% RSLogix 500 project CANHOES E PERFURATRIZES 1.RSS, saved by version 10.00.00.00 %
PROJECT "USIMINAS"    % processor: SLC 500, 1747-L552 %

PROGRAM FILES
  LAD 2 "PRINCIPAL"  17 rungs
  LAD 5 "ANA OUT"  17 rungs  % Bloco de transferencia do 1746-NO4V para o SCANNER %
  LAD 7 "BOMBA 1"  25 rungs  % Bomba 1 %
  LAD 8 "BOMBA 2"  21 rungs  % Bomba 2 %
  LAD 9 "BOMBA REF"  17 rungs  % Bomba Refrigeracao 1 %
  LAD 11 "PRESS INJ"  7 rungs  % Pressao de injecao mais alta %
  LAD 12 "TRACO INJ"  11 rungs  % Volume Lama Injetado %
  LAD 13 "CANHAO"  24 rungs  % Controle do Giro do Canhao %
  LAD 14 "INJECAO M"  10 rungs
  LAD 15 "PERFURAT"  29 rungs
  LAD 16 "MARTELETE"  10 rungs
  LAD 17 "BOMBA AGUA"  15 rungs  % Resfriamento da Broca ou Sopro %
  LAD 18 "ALR GERAIS"  69 rungs  % ALARMES GERAIS E ANUNCIADOR %
  LAD 19 "COMUNIC"  20 rungs  % Comuinicao com supervisorio - Desabilitado(futuro) %
  LAD 20 "HISTERESE"  6 rungs
  LAD 21 "ALR ANALOG"  70 rungs  % Alarmes Analogicos %
  LAD 22 "UNID ENG"  20 rungs
  LAD 23 "RESET"  10 rungs  % Reset geral para 1 scan %

DATA FILES
  O0 OUTPUT  52 elements
  I1 INPUT  46 elements
  S2 STATUS  83 elements
  B3 BINARY  63 elements
  T4 TIMER  201 elements
  C5 COUNTER  1 elements
  R6 CONTROL  4 elements
  N7 INTEGER  3 elements
  F8 FLOAT  50 elements
  B9 COMANDO D  28 elements
  B10 ESPELHO D  16 elements  % Area Espelho entradas e saidas digitais %
  B11 STATUS  68 elements  % Status do sistema que são enviados ao SSC %
  B13 DEFEITO  112 elements
  N15 ESPELHO A  50 elements  % Area Espelho entradas e saidas analogicas %
  N16 SET POINT  90 elements
  N17 LEITURA  90 elements
  N18 COMANDO A  1 elements  % Comando Analogico %
  B20 ESPELHO O  12 elements
  B21 AUXILIARES  20 elements  % auxiliares %
  B22   1 elements
  B23   1 elements
  N24 SAIDAS ANA  20 elements
  N25 B TRANSFER  10 elements  % Utilizado pelo Bloco Transfer %
  N26 COM SUP  51 elements  % Area para comunicacao com Supervisorio %
  N27 COM SUP  51 elements  % Area para comunicacao com Supervisorio %
  N29 HISTERESE  9 elements  % Valores para calculo de histerese %
  B31 AUX STATUS  26 elements
  B33 AUX DEF  26 elements
  B39 LEIT SUP  10 elements  % Area de mensagens que sao enviadas ao Supervisorio %
  B40 LEIT SUP  10 elements  % Area de mensagens que sao enviadas ao Supervisorio %
  B41 LEIT SUP  8 elements  % Area de mensagens que sao enviadas ao Supervisorio %
  B42 LEIT SUP  1 elements  % Area de mensagens que sao enviadas ao Supervisorio %

LADDER 2 "PRINCIPAL"
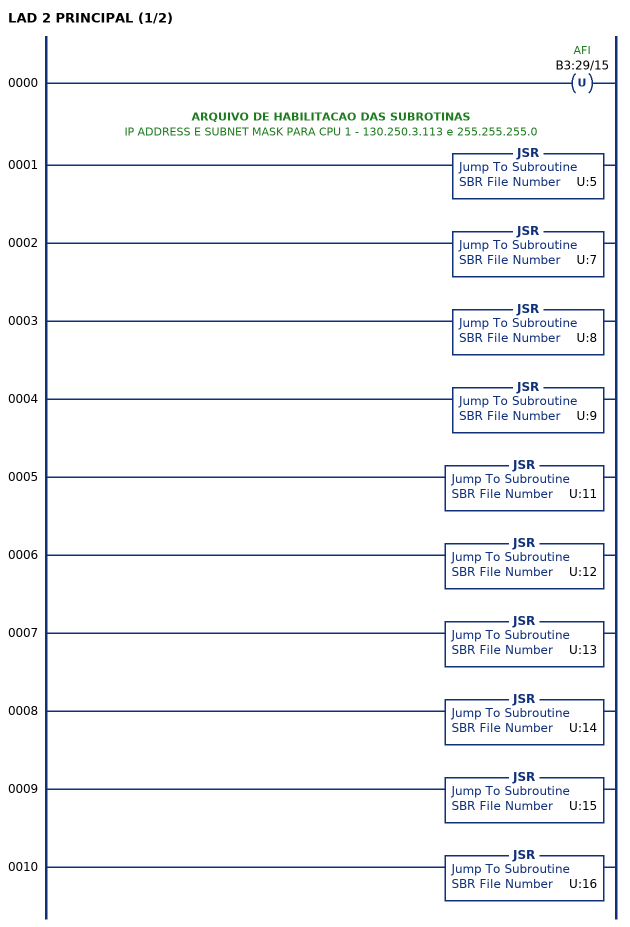
% Rung: 0 %
SOR OTU B3:29/15 EOR
%   B3:29/15  AFI %
% Rung: 1 %
% TITLE: ARQUIVO DE HABILITACAO DAS SUBROTINAS %
% IP ADDRESS E SUBNET MASK PARA CPU 1 - 130.250.3.113 e 255.255.255.0 %
SOR JSR U:5 EOR
% Rung: 2 %
SOR JSR U:7 EOR
% Rung: 3 %
SOR JSR U:8 EOR
% Rung: 4 %
SOR JSR U:9 EOR
% Rung: 5 %
SOR JSR U:11 EOR
% Rung: 6 %
SOR JSR U:12 EOR
% Rung: 7 %
SOR JSR U:13 EOR
% Rung: 8 %
SOR JSR U:14 EOR
% Rung: 9 %
SOR JSR U:15 EOR
% Rung: 10 %
SOR JSR U:16 EOR

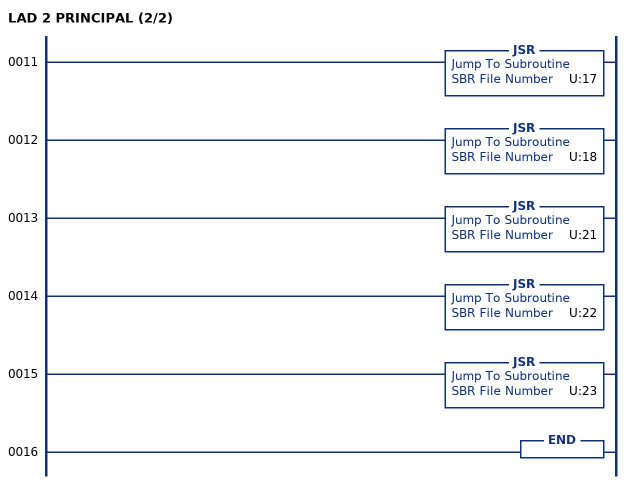
% Rung: 11 %
SOR JSR U:17 EOR
% Rung: 12 %
SOR JSR U:18 EOR
% Rung: 13 %
SOR JSR U:21 EOR
% Rung: 14 %
SOR JSR U:22 EOR
% Rung: 15 %
SOR JSR U:23 EOR
% Rung: 16 %
SOR END EOR

LADDER 5 "ANA OUT"    % Bloco de transferencia do 1746-NO4V para o SCANNER %
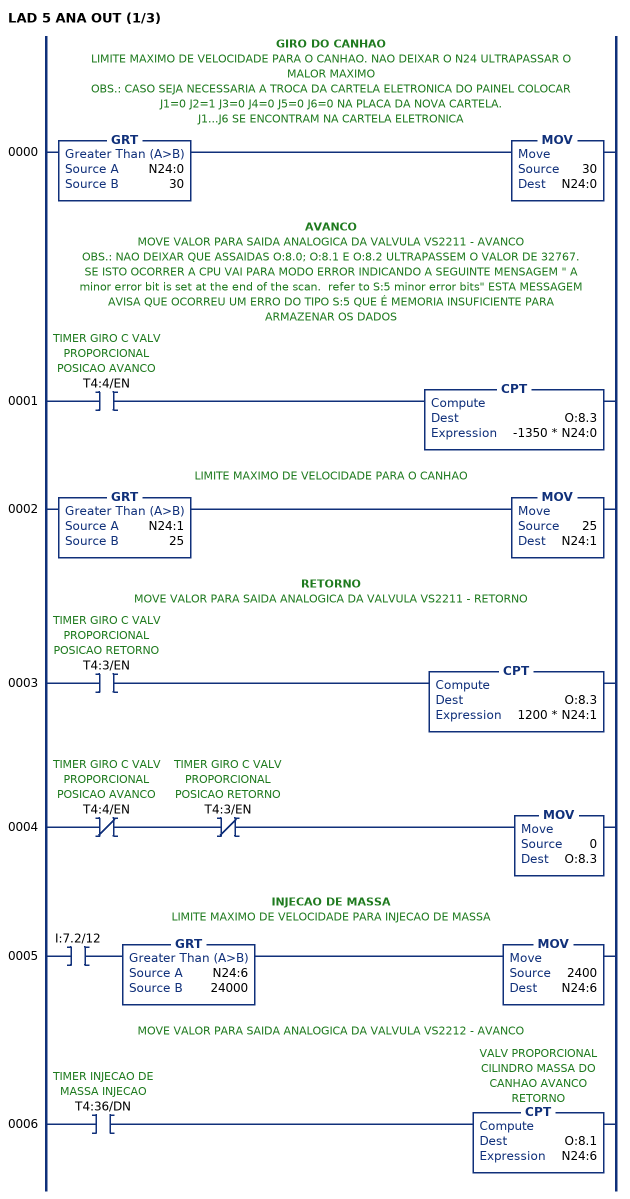
% Rung: 0 %
% TITLE: GIRO DO CANHAO %
% LIMITE MAXIMO DE VELOCIDADE PARA O CANHAO. NAO DEIXAR O N24 ULTRAPASSAR O MALOR MAXIMO
% OBS.: CASO SEJA NECESSARIA A TROCA DA CARTELA ELETRONICA DO PAINEL COLOCAR
% J1=0 J2=1 J3=0 J4=0 J5=0 J6=0 NA PLACA DA NOVA CARTELA.
% J1...J6 SE ENCONTRAM NA CARTELA ELETRONICA %
SOR GRT N24:0 30 MOV 30 N24:0 EOR
% Rung: 1 %
% TITLE: AVANCO %
% MOVE VALOR PARA SAIDA ANALOGICA DA VALVULA VS2211 - AVANCO
% OBS.: NAO DEIXAR QUE ASSAIDAS O:8.0; O:8.1 E O:8.2 ULTRAPASSEM O VALOR DE 32767. SE ISTO OCORRER A CPU VAI PARA MODO ERROR INDICANDO A SEGUINTE MENSAGEM " A minor error bit is set at the end of the scan.  refer to S:5 minor error bits" ESTA MESSAGEM AVISA QUE OCORREU UM ERRO DO TIPO S:5 QUE É MEMORIA INSUFICIENTE PARA ARMAZENAR OS DADOS %
SOR XIC T4:4/EN CPT O:8.3 " -1350 * N24:0 " EOR
%   T4:4  "TIMER GIRO C VALV PROPORCIONAL POSICAO AVANCO" %
% Rung: 2 %
% LIMITE MAXIMO DE VELOCIDADE PARA O CANHAO %
SOR GRT N24:1 25 MOV 25 N24:1 EOR
% Rung: 3 %
% TITLE: RETORNO %
% MOVE VALOR PARA SAIDA ANALOGICA DA VALVULA VS2211 - RETORNO %
SOR XIC T4:3/EN CPT O:8.3 " 1200 * N24:1 " EOR
%   T4:3  "TIMER GIRO C VALV PROPORCIONAL POSICAO RETORNO" %
% Rung: 4 %
SOR XIO T4:4/EN XIO T4:3/EN MOV 0 O:8.3 EOR
%   T4:4  "TIMER GIRO C VALV PROPORCIONAL POSICAO AVANCO" %
%   T4:3  "TIMER GIRO C VALV PROPORCIONAL POSICAO RETORNO" %
% Rung: 5 %
% TITLE: INJECAO DE MASSA %
% LIMITE MAXIMO DE VELOCIDADE PARA INJECAO DE MASSA %
SOR XIC I:7.2/12 GRT N24:6 24000 MOV 2400 N24:6 EOR
% Rung: 6 %
% MOVE VALOR PARA SAIDA ANALOGICA DA VALVULA VS2212 - AVANCO %
SOR XIC T4:36/DN CPT O:8.1 "  N24:6 " EOR
%   T4:36  "TIMER INJECAO DE MASSA INJECAO" %
%   O:8.1  "VALV PROPORCIONAL CILINDRO MASSA DO CANHAO AVANCO RETORNO" %

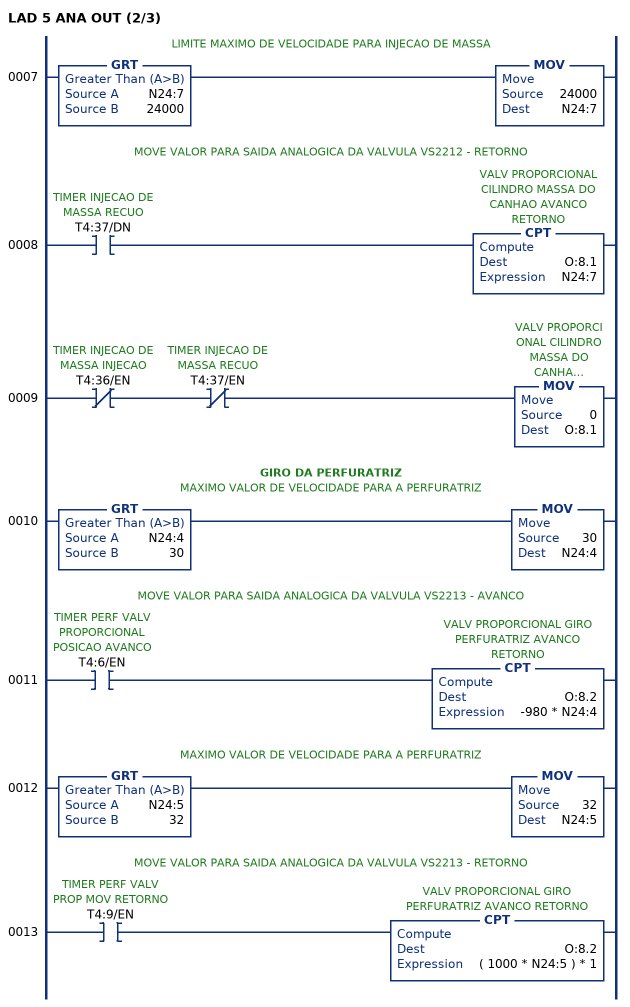
% Rung: 7 %
% LIMITE MAXIMO DE VELOCIDADE PARA INJECAO DE MASSA %
SOR GRT N24:7 24000 MOV 24000 N24:7 EOR
% Rung: 8 %
% MOVE VALOR PARA SAIDA ANALOGICA DA VALVULA VS2212 - RETORNO %
SOR XIC T4:37/DN CPT O:8.1 "  N24:7 " EOR
%   T4:37  "TIMER INJECAO DE MASSA RECUO" %
%   O:8.1  "VALV PROPORCIONAL CILINDRO MASSA DO CANHAO AVANCO RETORNO" %
% Rung: 9 %
SOR XIO T4:36/EN XIO T4:37/EN MOV 0 O:8.1 EOR
%   T4:36  "TIMER INJECAO DE MASSA INJECAO" %
%   T4:37  "TIMER INJECAO DE MASSA RECUO" %
%   O:8.1  "VALV PROPORCIONAL CILINDRO MASSA DO CANHAO AVANCO RETORNO" %
% Rung: 10 %
% TITLE: GIRO DA PERFURATRIZ %
% MAXIMO VALOR DE VELOCIDADE PARA A PERFURATRIZ %
SOR GRT N24:4 30 MOV 30 N24:4 EOR
% Rung: 11 %
% MOVE VALOR PARA SAIDA ANALOGICA DA VALVULA VS2213 - AVANCO %
SOR XIC T4:6/EN CPT O:8.2 " -980 * N24:4 " EOR
%   T4:6  "TIMER PERF VALV PROPORCIONAL POSICAO AVANCO" %
%   O:8.2  "VALV PROPORCIONAL GIRO PERFURATRIZ AVANCO RETORNO" %
% Rung: 12 %
% MAXIMO VALOR DE VELOCIDADE PARA A PERFURATRIZ %
SOR GRT N24:5 32 MOV 32 N24:5 EOR
% Rung: 13 %
% MOVE VALOR PARA SAIDA ANALOGICA DA VALVULA VS2213 - RETORNO %
SOR XIC T4:9/EN CPT O:8.2 " ( 1000 * N24:5 ) * 1 " EOR
%   T4:9  "TIMER PERF VALV PROP MOV RETORNO" %
%   O:8.2  "VALV PROPORCIONAL GIRO PERFURATRIZ AVANCO RETORNO" %

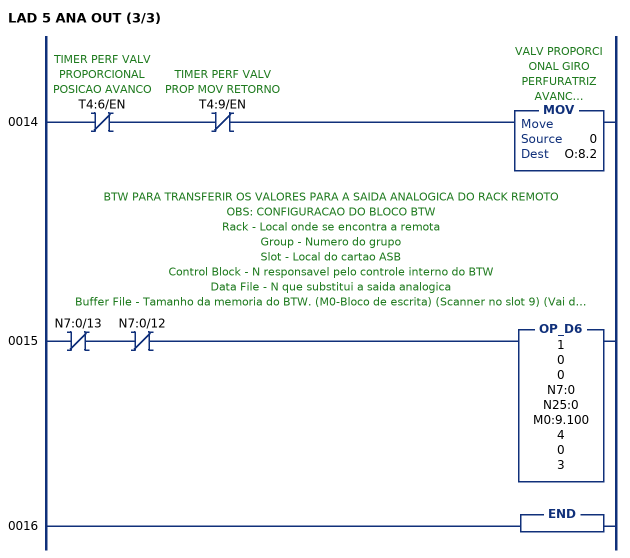
% Rung: 14 %
SOR XIO T4:6/EN XIO T4:9/EN MOV 0 O:8.2 EOR
%   T4:6  "TIMER PERF VALV PROPORCIONAL POSICAO AVANCO" %
%   T4:9  "TIMER PERF VALV PROP MOV RETORNO" %
%   O:8.2  "VALV PROPORCIONAL GIRO PERFURATRIZ AVANCO RETORNO" %
% Rung: 15 %
% BTW PARA TRANSFERIR OS VALORES PARA A SAIDA ANALOGICA DO RACK REMOTO
% OBS: CONFIGURACAO DO BLOCO BTW
% Rack - Local onde se encontra a remota
% Group - Numero do grupo
% Slot - Local do cartao ASB
% Control Block - N responsavel pelo controle interno do BTW
% Data File - N que substitui a saida analogica
% Buffer File - Tamanho da memoria do BTW. (M0-Bloco de escrita) (Scanner no slot 9) (Vai de 100 a 3200)
% Req W. C - Quantidade de palavras usadas
% Trans. W. C. - Uso interno do BTW
% Control B. L - Uso interno do BTW %
SOR XIO N7:0/13 XIO N7:0/12 OP_D6 1 0 0 N7:0 N25:0 M0:9.100 4 0 3 EOR
% Rung: 16 %
SOR END EOR

LADDER 7 "BOMBA 1"    % Bomba 1 %
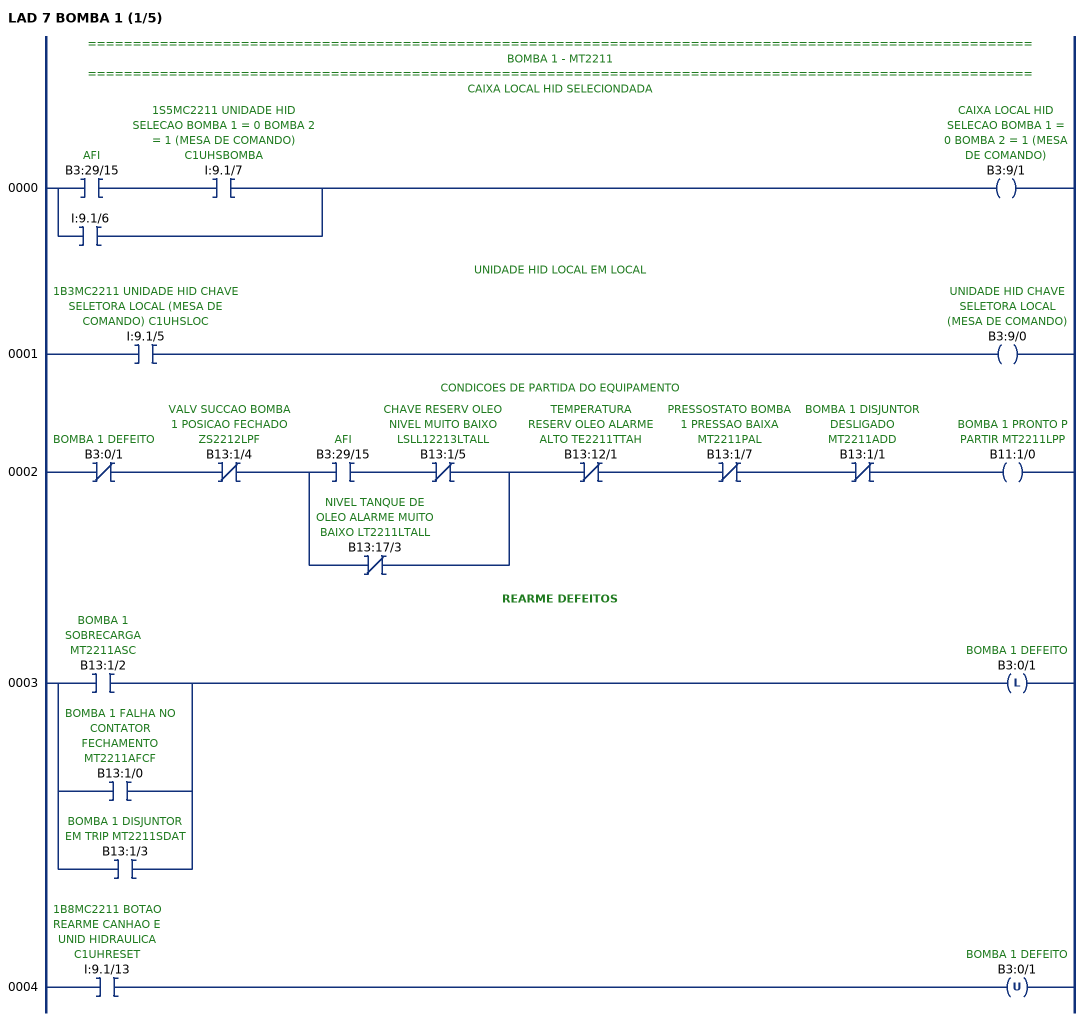
% Rung: 0 %
% =========================================================================================================
% BOMBA 1 - MT2211
% =========================================================================================================
% 
% CAIXA LOCAL HID SELECIONDADA %
SOR BST XIC B3:29/15 XIC I:9.1/7 NXB XIC I:9.1/6 BND OTE B3:9/1 EOR
%   B3:29/15  AFI %
%   I:9.1/7  C1UHSBOMBA  "1S5MC2211 UNIDADE HID SELECAO BOMBA 1 = 0 BOMBA 2 = 1 (MESA DE COMANDO)" %
%   B3:9/1  "CAIXA LOCAL HID SELECAO BOMBA 1 = 0 BOMBA 2 = 1 (MESA DE COMANDO)" %
% Rung: 1 %
% UNIDADE HID LOCAL EM LOCAL %
SOR XIC I:9.1/5 OTE B3:9/0 EOR
%   I:9.1/5  C1UHSLOC  "1B3MC2211 UNIDADE HID CHAVE SELETORA LOCAL (MESA DE COMANDO)" %
%   B3:9/0  "UNIDADE HID CHAVE SELETORA LOCAL (MESA DE COMANDO)" %
% Rung: 2 %
% CONDICOES DE PARTIDA DO EQUIPAMENTO %
SOR XIO B3:0/1 XIO B13:1/4 BST XIC B3:29/15 XIO B13:1/5 NXB XIO B13:17/3 BND XIO B13:12/1 XIO B13:1/7 XIO B13:1/1 OTE B11:1/0 EOR
%   B3:0/1  "BOMBA 1 DEFEITO" %
%   B13:1/4  ZS2212LPF  "VALV SUCCAO BOMBA 1 POSICAO FECHADO" %
%   B3:29/15  AFI %
%   B13:1/5  LSLL12213LTALL  "CHAVE RESERV OLEO NIVEL MUITO BAIXO" %
%   B13:17/3  LT2211LTALL  "NIVEL TANQUE DE OLEO ALARME MUITO BAIXO" %
%   B13:12/1  TE2211TTAH  "TEMPERATURA RESERV OLEO ALARME ALTO" %
%   B13:1/7  MT2211PAL  "PRESSOSTATO BOMBA 1 PRESSAO BAIXA" %
%   B13:1/1  MT2211ADD  "BOMBA 1 DISJUNTOR DESLIGADO" %
%   B11:1/0  MT2211LPP  "BOMBA 1 PRONTO P PARTIR" %
% Rung: 3 %
% TITLE: REARME DEFEITOS %
SOR BST XIC B13:1/2 NXB XIC B13:1/0 NXB XIC B13:1/3 BND OTL B3:0/1 EOR
%   B13:1/2  MT2211ASC  "BOMBA 1 SOBRECARGA" %
%   B13:1/0  MT2211AFCF  "BOMBA 1 FALHA NO CONTATOR FECHAMENTO" %
%   B13:1/3  MT2211SDAT  "BOMBA 1 DISJUNTOR EM TRIP" %
%   B3:0/1  "BOMBA 1 DEFEITO" %
% Rung: 4 %
SOR XIC I:9.1/13 OTU B3:0/1 EOR
%   I:9.1/13  C1UHRESET  "1B8MC2211 BOTAO REARME CANHAO E UNID HIDRAULICA" %
%   B3:0/1  "BOMBA 1 DEFEITO" %

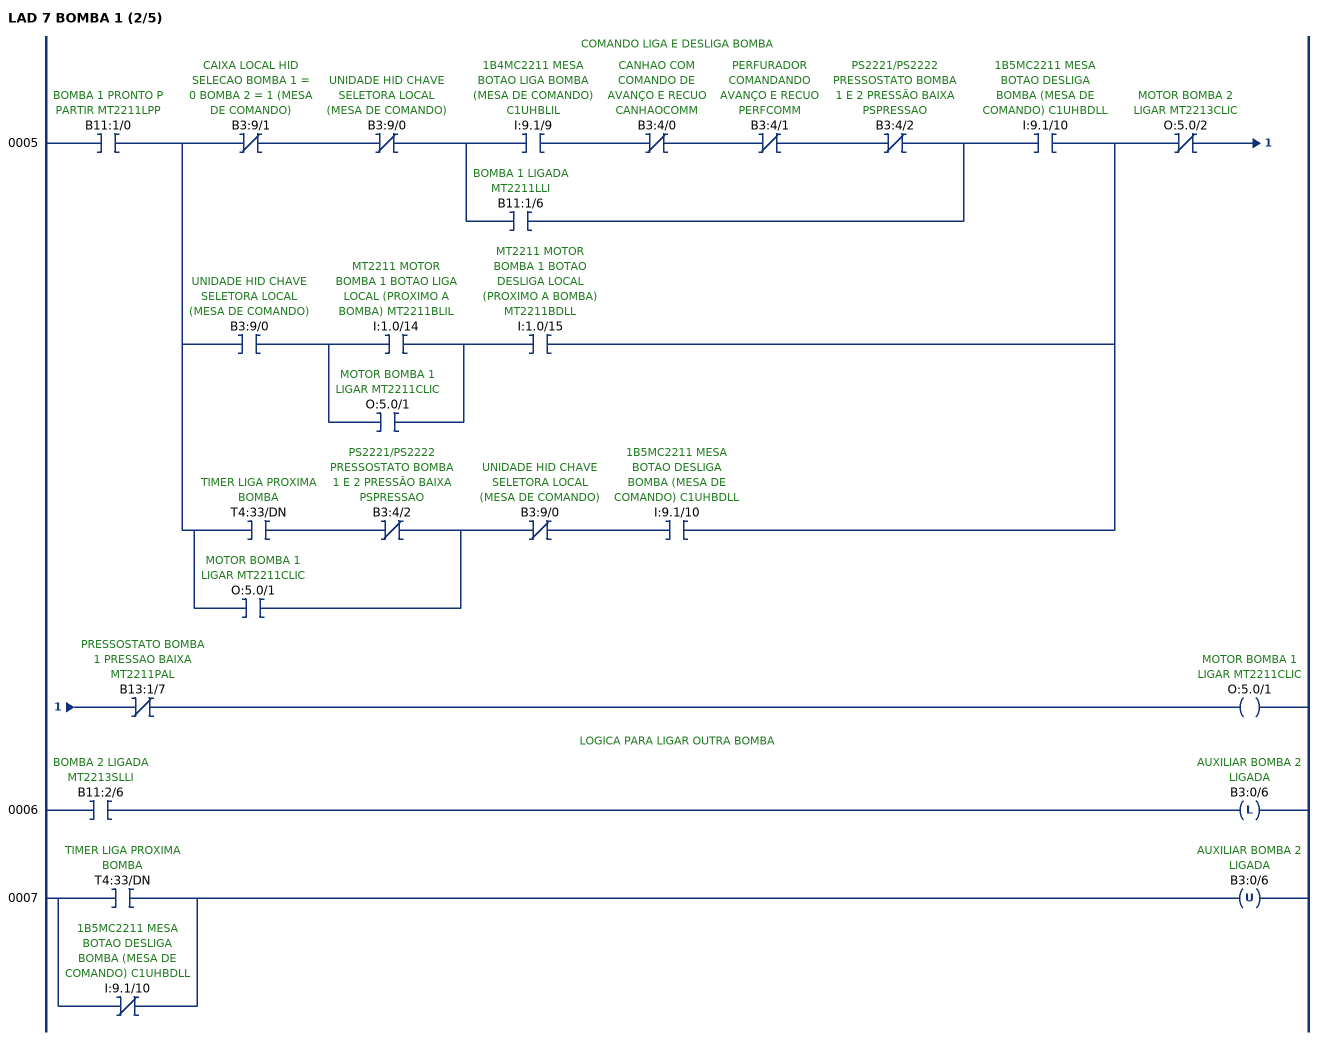
% Rung: 5 %
% COMANDO LIGA E DESLIGA BOMBA %
SOR XIC B11:1/0 BST XIO B3:9/1 XIO B3:9/0 BST XIC I:9.1/9 XIO B3:4/0 XIO B3:4/1 XIO B3:4/2 NXB XIC B11:1/6 BND XIC I:9.1/10 NXB XIC B3:9/0 BST XIC I:1.0/14 NXB XIC O:5.0/1 BND XIC I:1.0/15 NXB BST XIC T4:33/DN XIO B3:4/2 NXB XIC O:5.0/1 BND XIO B3:9/0 XIC I:9.1/10 BND XIO O:5.0/2 XIO B13:1/7 OTE O:5.0/1 EOR
%   B11:1/0  MT2211LPP  "BOMBA 1 PRONTO P PARTIR" %
%   B3:9/1  "CAIXA LOCAL HID SELECAO BOMBA 1 = 0 BOMBA 2 = 1 (MESA DE COMANDO)" %
%   B3:9/0  "UNIDADE HID CHAVE SELETORA LOCAL (MESA DE COMANDO)" %
%   I:9.1/9  C1UHBLIL  "1B4MC2211 MESA BOTAO LIGA BOMBA (MESA DE COMANDO)" %
%   B3:4/0  CANHAOCOMM  "CANHAO COM COMANDO DE AVANÇO E RECUO" %
%   B3:4/1  PERFCOMM  "PERFURADOR COMANDANDO AVANÇO E RECUO" %
%   B3:4/2  PSPRESSAO  "PS2221/PS2222 PRESSOSTATO BOMBA 1 E 2 PRESSÃO BAIXA" %
%   B11:1/6  MT2211LLI  "BOMBA 1 LIGADA" %
%   I:9.1/10  C1UHBDLL  "1B5MC2211 MESA BOTAO DESLIGA BOMBA (MESA DE COMANDO)" %
%   I:1.0/14  MT2211BLIL  "MT2211 MOTOR BOMBA 1 BOTAO LIGA LOCAL (PROXIMO A BOMBA)" %
%   O:5.0/1  MT2211CLIC  "MOTOR BOMBA 1 LIGAR" %
%   I:1.0/15  MT2211BDLL  "MT2211 MOTOR BOMBA 1 BOTAO DESLIGA LOCAL (PROXIMO A BOMBA)" %
%   T4:33  "TIMER LIGA PROXIMA BOMBA" %
%   O:5.0/2  MT2213CLIC  "MOTOR BOMBA 2 LIGAR" %
%   B13:1/7  MT2211PAL  "PRESSOSTATO BOMBA 1 PRESSAO BAIXA" %
% Rung: 6 %
% LOGICA PARA LIGAR OUTRA BOMBA %
SOR XIC B11:2/6 OTL B3:0/6 EOR
%   B11:2/6  MT2213SLLI  "BOMBA 2 LIGADA" %
%   B3:0/6  "AUXILIAR BOMBA 2 LIGADA" %
% Rung: 7 %
SOR BST XIC T4:33/DN NXB XIO I:9.1/10 BND OTU B3:0/6 EOR
%   T4:33  "TIMER LIGA PROXIMA BOMBA" %
%   I:9.1/10  C1UHBDLL  "1B5MC2211 MESA BOTAO DESLIGA BOMBA (MESA DE COMANDO)" %
%   B3:0/6  "AUXILIAR BOMBA 2 LIGADA" %

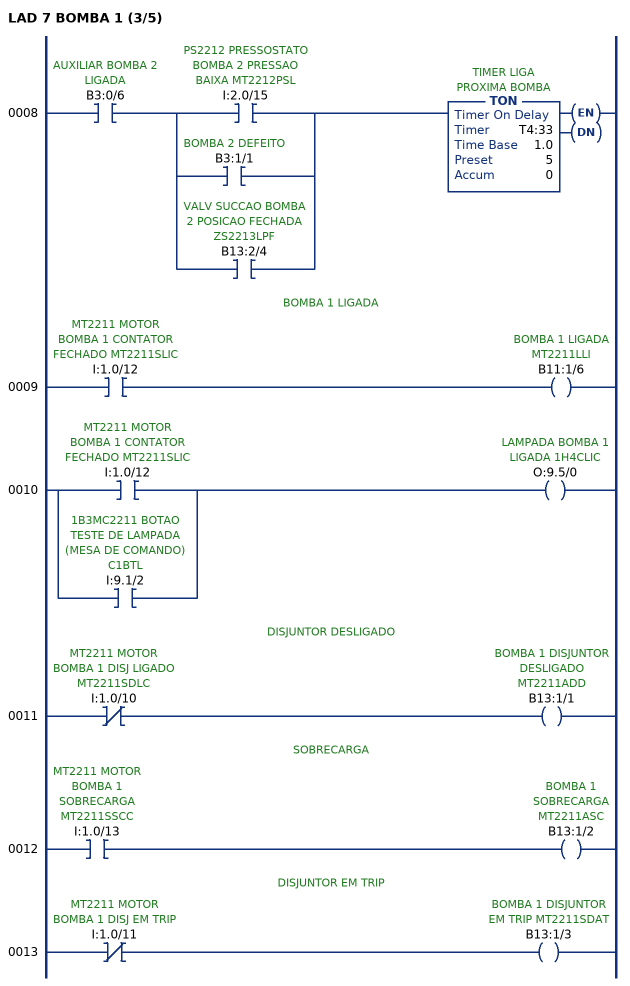
% Rung: 8 %
SOR XIC B3:0/6 BST XIC I:2.0/15 NXB XIC B3:1/1 NXB XIC B13:2/4 BND TON T4:33 1.0 5 0 EOR
%   B3:0/6  "AUXILIAR BOMBA 2 LIGADA" %
%   I:2.0/15  MT2212PSL  "PS2212 PRESSOSTATO BOMBA 2 PRESSAO BAIXA" %
%   B3:1/1  "BOMBA 2 DEFEITO" %
%   B13:2/4  ZS2213LPF  "VALV SUCCAO BOMBA 2 POSICAO FECHADA" %
%   T4:33  "TIMER LIGA PROXIMA BOMBA" %
% Rung: 9 %
% BOMBA 1 LIGADA %
SOR XIC I:1.0/12 OTE B11:1/6 EOR
%   I:1.0/12  MT2211SLIC  "MT2211 MOTOR BOMBA 1 CONTATOR FECHADO" %
%   B11:1/6  MT2211LLI  "BOMBA 1 LIGADA" %
% Rung: 10 %
SOR BST XIC I:1.0/12 NXB XIC I:9.1/2 BND OTE O:9.5/0 EOR
%   I:1.0/12  MT2211SLIC  "MT2211 MOTOR BOMBA 1 CONTATOR FECHADO" %
%   I:9.1/2  C1BTL  "1B3MC2211 BOTAO TESTE DE LAMPADA (MESA DE COMANDO)" %
%   O:9.5/0  1H4CLIC  "LAMPADA BOMBA 1 LIGADA" %
% Rung: 11 %
% DISJUNTOR DESLIGADO %
SOR XIO I:1.0/10 OTE B13:1/1 EOR
%   I:1.0/10  MT2211SDLC  "MT2211 MOTOR BOMBA 1 DISJ LIGADO" %
%   B13:1/1  MT2211ADD  "BOMBA 1 DISJUNTOR DESLIGADO" %
% Rung: 12 %
% SOBRECARGA %
SOR XIC I:1.0/13 OTE B13:1/2 EOR
%   I:1.0/13  MT2211SSCC  "MT2211 MOTOR BOMBA 1 SOBRECARGA" %
%   B13:1/2  MT2211ASC  "BOMBA 1 SOBRECARGA" %
% Rung: 13 %
% DISJUNTOR EM TRIP %
SOR XIO I:1.0/11 OTE B13:1/3 EOR
%   I:1.0/11  "MT2211 MOTOR BOMBA 1 DISJ EM TRIP" %
%   B13:1/3  MT2211SDAT  "BOMBA 1 DISJUNTOR EM TRIP" %

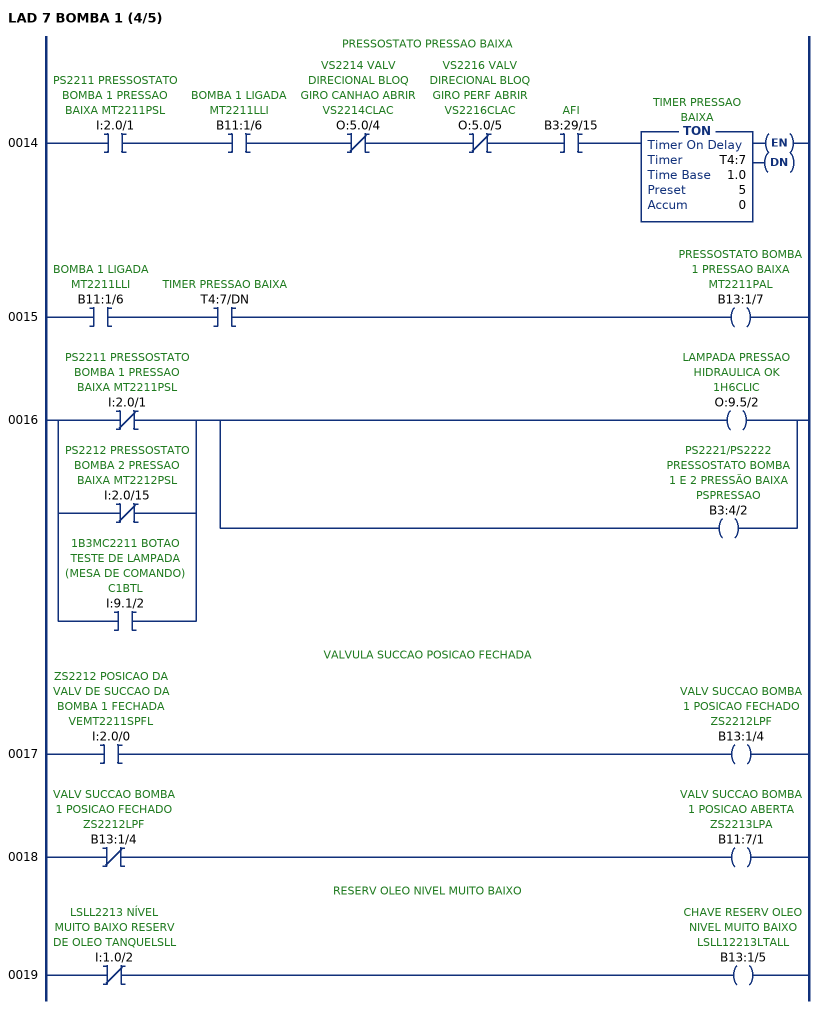
% Rung: 14 %
% PRESSOSTATO PRESSAO BAIXA %
SOR XIC I:2.0/1 XIC B11:1/6 XIO O:5.0/4 XIO O:5.0/5 XIC B3:29/15 TON T4:7 1.0 5 0 EOR
%   I:2.0/1  MT2211PSL  "PS2211 PRESSOSTATO BOMBA 1 PRESSAO BAIXA" %
%   B11:1/6  MT2211LLI  "BOMBA 1 LIGADA" %
%   O:5.0/4  VS2214CLAC  "VS2214 VALV DIRECIONAL BLOQ GIRO CANHAO ABRIR" %
%   O:5.0/5  VS2216CLAC  "VS2216 VALV DIRECIONAL BLOQ GIRO PERF ABRIR" %
%   B3:29/15  AFI %
%   T4:7  "TIMER PRESSAO BAIXA" %
% Rung: 15 %
SOR XIC B11:1/6 XIC T4:7/DN OTE B13:1/7 EOR
%   B11:1/6  MT2211LLI  "BOMBA 1 LIGADA" %
%   T4:7  "TIMER PRESSAO BAIXA" %
%   B13:1/7  MT2211PAL  "PRESSOSTATO BOMBA 1 PRESSAO BAIXA" %
% Rung: 16 %
SOR BST XIO I:2.0/1 NXB XIO I:2.0/15 NXB XIC I:9.1/2 BND BST OTE O:9.5/2 NXB OTE B3:4/2 BND EOR
%   I:2.0/1  MT2211PSL  "PS2211 PRESSOSTATO BOMBA 1 PRESSAO BAIXA" %
%   I:2.0/15  MT2212PSL  "PS2212 PRESSOSTATO BOMBA 2 PRESSAO BAIXA" %
%   I:9.1/2  C1BTL  "1B3MC2211 BOTAO TESTE DE LAMPADA (MESA DE COMANDO)" %
%   O:9.5/2  1H6CLIC  "LAMPADA PRESSAO HIDRAULICA OK" %
%   B3:4/2  PSPRESSAO  "PS2221/PS2222 PRESSOSTATO BOMBA 1 E 2 PRESSÃO BAIXA" %
% Rung: 17 %
% VALVULA SUCCAO POSICAO FECHADA %
SOR XIC I:2.0/0 OTE B13:1/4 EOR
%   I:2.0/0  VEMT2211SPFL  "ZS2212 POSICAO DA VALV DE SUCCAO DA BOMBA 1 FECHADA" %
%   B13:1/4  ZS2212LPF  "VALV SUCCAO BOMBA 1 POSICAO FECHADO" %
% Rung: 18 %
SOR XIO B13:1/4 OTE B11:7/1 EOR
%   B13:1/4  ZS2212LPF  "VALV SUCCAO BOMBA 1 POSICAO FECHADO" %
%   B11:7/1  ZS2213LPA  "VALV SUCCAO BOMBA 1 POSICAO ABERTA" %
% Rung: 19 %
% RESERV OLEO NIVEL MUITO BAIXO %
SOR XIO I:1.0/2 OTE B13:1/5 EOR
%   I:1.0/2  TANQUELSLL  "LSLL2213 NÍVEL MUITO BAIXO RESERV DE OLEO" %
%   B13:1/5  LSLL12213LTALL  "CHAVE RESERV OLEO NIVEL MUITO BAIXO" %

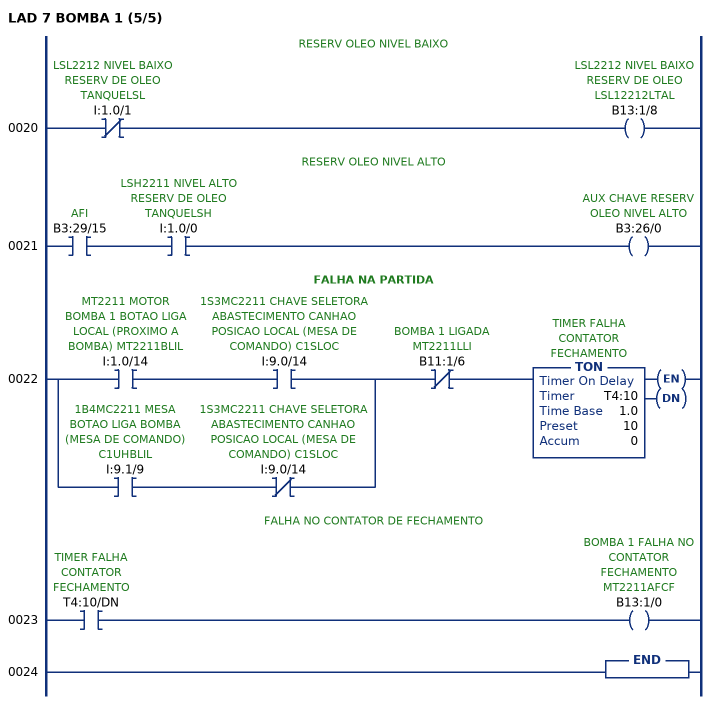
% Rung: 20 %
% RESERV OLEO NIVEL BAIXO %
SOR XIO I:1.0/1 OTE B13:1/8 EOR
%   I:1.0/1  TANQUELSL  "LSL2212 NIVEL BAIXO RESERV DE OLEO" %
%   B13:1/8  LSL12212LTAL  "LSL2212 NIVEL BAIXO RESERV DE OLEO" %
% Rung: 21 %
% RESERV OLEO NIVEL ALTO %
SOR XIC B3:29/15 XIC I:1.0/0 OTE B3:26/0 EOR
%   B3:29/15  AFI %
%   I:1.0/0  TANQUELSH  "LSH2211 NIVEL ALTO RESERV DE OLEO" %
%   B3:26/0  "AUX CHAVE RESERV OLEO NIVEL ALTO" %
% Rung: 22 %
% TITLE: FALHA NA PARTIDA %
SOR BST XIC I:1.0/14 XIC I:9.0/14 NXB XIC I:9.1/9 XIO I:9.0/14 BND XIO B11:1/6 TON T4:10 1.0 10 0 EOR
%   I:1.0/14  MT2211BLIL  "MT2211 MOTOR BOMBA 1 BOTAO LIGA LOCAL (PROXIMO A BOMBA)" %
%   I:9.0/14  C1SLOC  "1S3MC2211 CHAVE SELETORA ABASTECIMENTO CANHAO POSICAO LOCAL (MESA DE COMANDO)" %
%   I:9.1/9  C1UHBLIL  "1B4MC2211 MESA BOTAO LIGA BOMBA (MESA DE COMANDO)" %
%   B11:1/6  MT2211LLI  "BOMBA 1 LIGADA" %
%   T4:10  "TIMER FALHA CONTATOR FECHAMENTO" %
% Rung: 23 %
% FALHA NO CONTATOR DE FECHAMENTO %
SOR XIC T4:10/DN OTE B13:1/0 EOR
%   T4:10/DN  "TIMER FALHA CONTATOR FECHAMENTO" %
%   B13:1/0  MT2211AFCF  "BOMBA 1 FALHA NO CONTATOR FECHAMENTO" %
% Rung: 24 %
SOR END EOR

LADDER 8 "BOMBA 2"    % Bomba 2 %
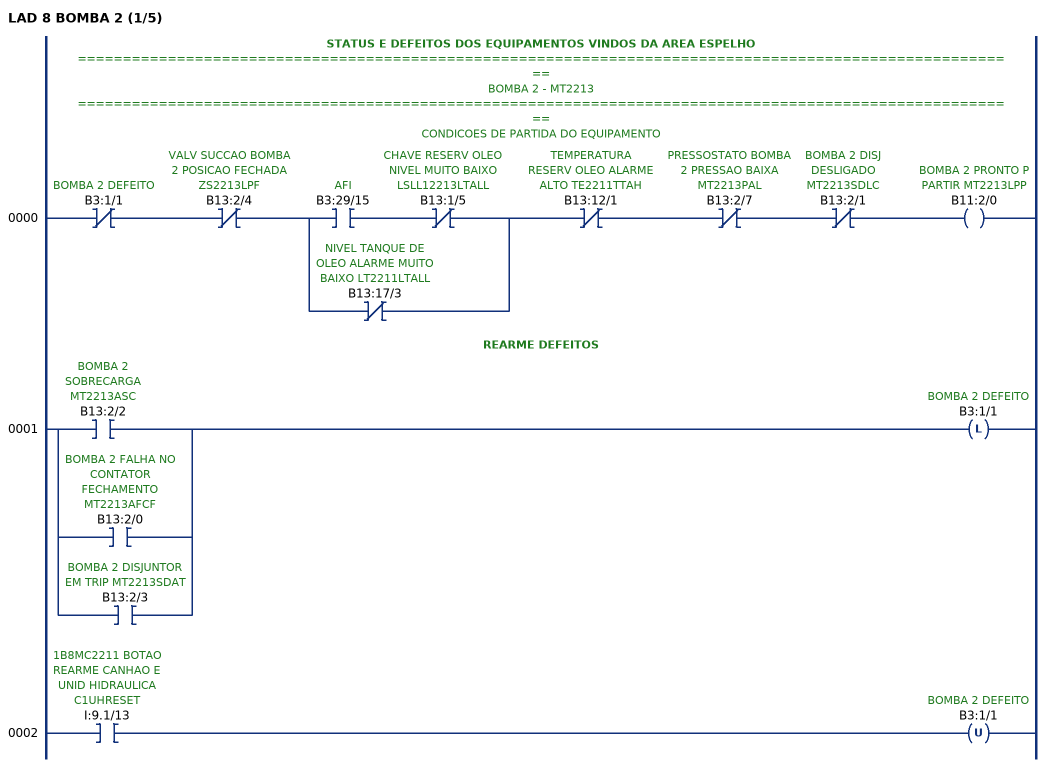
% Rung: 0 %
% TITLE: STATUS E DEFEITOS DOS EQUIPAMENTOS VINDOS DA AREA ESPELHO %
% =========================================================================================================
% BOMBA 2 - MT2213
% =========================================================================================================
% 
% CONDICOES DE PARTIDA DO EQUIPAMENTO %
SOR XIO B3:1/1 XIO B13:2/4 BST XIC B3:29/15 XIO B13:1/5 NXB XIO B13:17/3 BND XIO B13:12/1 XIO B13:2/7 XIO B13:2/1 OTE B11:2/0 EOR
%   B3:1/1  "BOMBA 2 DEFEITO" %
%   B13:2/4  ZS2213LPF  "VALV SUCCAO BOMBA 2 POSICAO FECHADA" %
%   B3:29/15  AFI %
%   B13:1/5  LSLL12213LTALL  "CHAVE RESERV OLEO NIVEL MUITO BAIXO" %
%   B13:17/3  LT2211LTALL  "NIVEL TANQUE DE OLEO ALARME MUITO BAIXO" %
%   B13:12/1  TE2211TTAH  "TEMPERATURA RESERV OLEO ALARME ALTO" %
%   B13:2/7  MT2213PAL  "PRESSOSTATO BOMBA 2 PRESSAO BAIXA" %
%   B13:2/1  MT2213SDLC  "BOMBA 2 DISJ DESLIGADO" %
%   B11:2/0  MT2213LPP  "BOMBA 2 PRONTO P PARTIR" %
% Rung: 1 %
% TITLE: REARME DEFEITOS %
SOR BST XIC B13:2/2 NXB XIC B13:2/0 NXB XIC B13:2/3 BND OTL B3:1/1 EOR
%   B13:2/2  MT2213ASC  "BOMBA 2 SOBRECARGA" %
%   B13:2/0  MT2213AFCF  "BOMBA 2 FALHA NO CONTATOR FECHAMENTO" %
%   B13:2/3  MT2213SDAT  "BOMBA 2 DISJUNTOR EM TRIP" %
%   B3:1/1  "BOMBA 2 DEFEITO" %
% Rung: 2 %
SOR XIC I:9.1/13 OTU B3:1/1 EOR
%   I:9.1/13  C1UHRESET  "1B8MC2211 BOTAO REARME CANHAO E UNID HIDRAULICA" %
%   B3:1/1  "BOMBA 2 DEFEITO" %

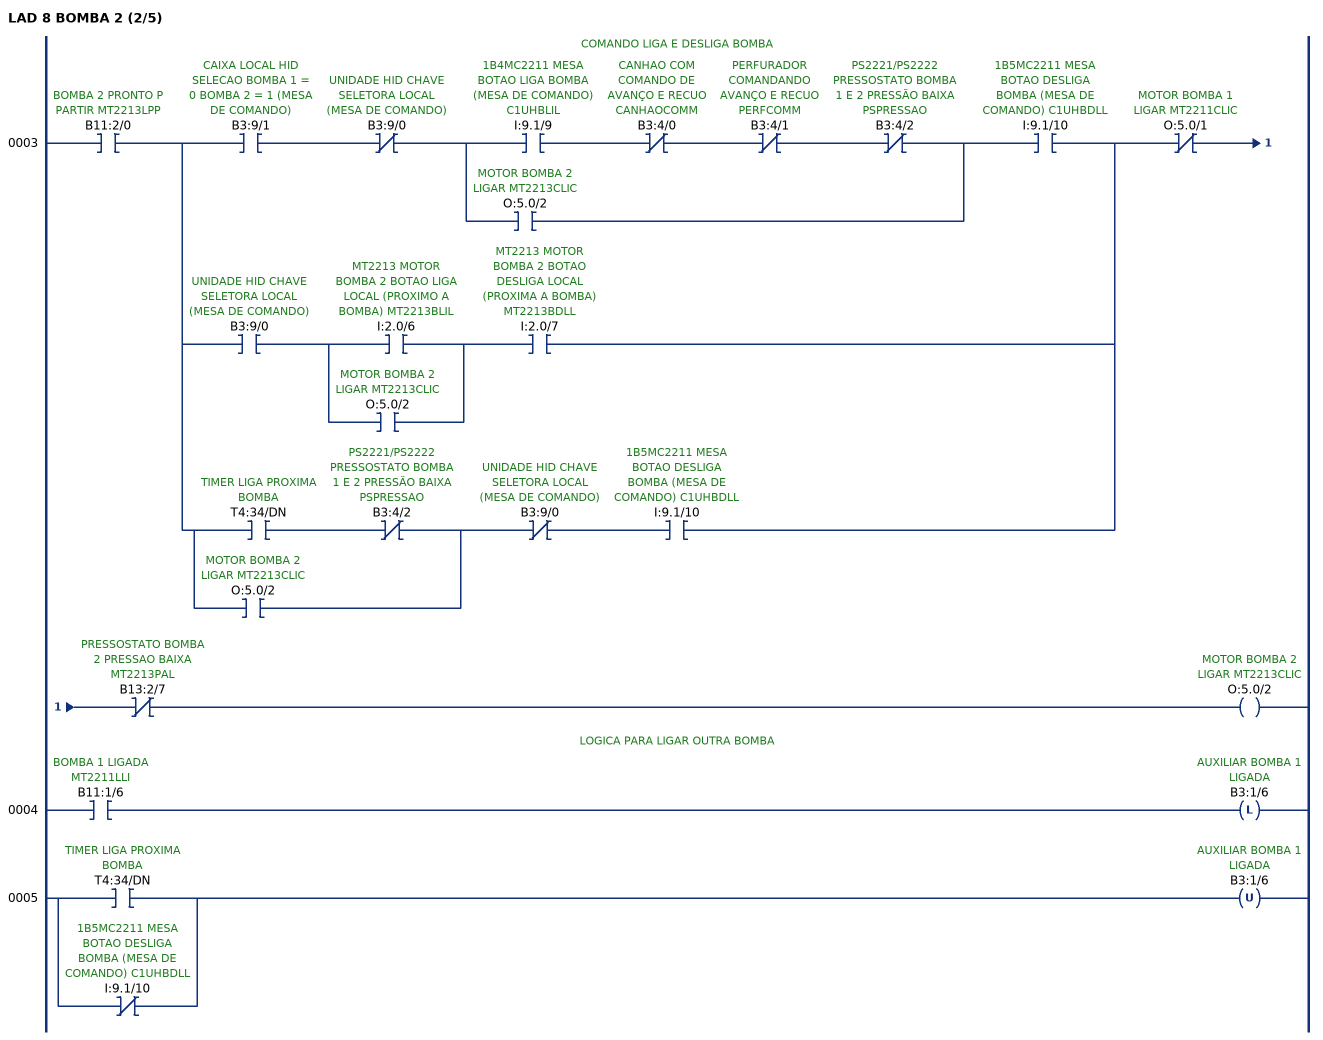
% Rung: 3 %
% COMANDO LIGA E DESLIGA BOMBA %
SOR XIC B11:2/0 BST XIC B3:9/1 XIO B3:9/0 BST XIC I:9.1/9 XIO B3:4/0 XIO B3:4/1 XIO B3:4/2 NXB XIC O:5.0/2 BND XIC I:9.1/10 NXB XIC B3:9/0 BST XIC I:2.0/6 NXB XIC O:5.0/2 BND XIC I:2.0/7 NXB BST XIC T4:34/DN XIO B3:4/2 NXB XIC O:5.0/2 BND XIO B3:9/0 XIC I:9.1/10 BND XIO O:5.0/1 XIO B13:2/7 OTE O:5.0/2 EOR
%   B11:2/0  MT2213LPP  "BOMBA 2 PRONTO P PARTIR" %
%   B3:9/1  "CAIXA LOCAL HID SELECAO BOMBA 1 = 0 BOMBA 2 = 1 (MESA DE COMANDO)" %
%   B3:9/0  "UNIDADE HID CHAVE SELETORA LOCAL (MESA DE COMANDO)" %
%   I:9.1/9  C1UHBLIL  "1B4MC2211 MESA BOTAO LIGA BOMBA (MESA DE COMANDO)" %
%   B3:4/0  CANHAOCOMM  "CANHAO COM COMANDO DE AVANÇO E RECUO" %
%   B3:4/1  PERFCOMM  "PERFURADOR COMANDANDO AVANÇO E RECUO" %
%   B3:4/2  PSPRESSAO  "PS2221/PS2222 PRESSOSTATO BOMBA 1 E 2 PRESSÃO BAIXA" %
%   O:5.0/2  MT2213CLIC  "MOTOR BOMBA 2 LIGAR" %
%   I:9.1/10  C1UHBDLL  "1B5MC2211 MESA BOTAO DESLIGA BOMBA (MESA DE COMANDO)" %
%   I:2.0/6  MT2213BLIL  "MT2213 MOTOR BOMBA 2 BOTAO LIGA LOCAL (PROXIMO A BOMBA)" %
%   I:2.0/7  MT2213BDLL  "MT2213 MOTOR BOMBA 2 BOTAO DESLIGA LOCAL (PROXIMA A BOMBA)" %
%   T4:34  "TIMER LIGA PROXIMA BOMBA" %
%   O:5.0/1  MT2211CLIC  "MOTOR BOMBA 1 LIGAR" %
%   B13:2/7  MT2213PAL  "PRESSOSTATO BOMBA 2 PRESSAO BAIXA" %
% Rung: 4 %
% LOGICA PARA LIGAR OUTRA BOMBA %
SOR XIC B11:1/6 OTL B3:1/6 EOR
%   B11:1/6  MT2211LLI  "BOMBA 1 LIGADA" %
%   B3:1/6  "AUXILIAR BOMBA 1 LIGADA" %
% Rung: 5 %
SOR BST XIC T4:34/DN NXB XIO I:9.1/10 BND OTU B3:1/6 EOR
%   T4:34  "TIMER LIGA PROXIMA BOMBA" %
%   I:9.1/10  C1UHBDLL  "1B5MC2211 MESA BOTAO DESLIGA BOMBA (MESA DE COMANDO)" %
%   B3:1/6  "AUXILIAR BOMBA 1 LIGADA" %

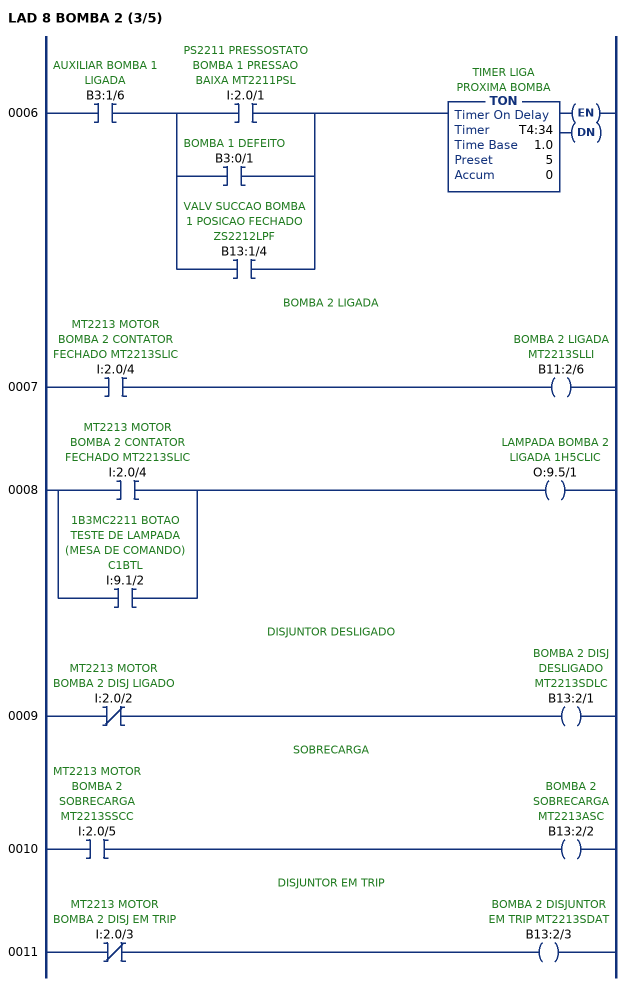
% Rung: 6 %
SOR XIC B3:1/6 BST XIC I:2.0/1 NXB XIC B3:0/1 NXB XIC B13:1/4 BND TON T4:34 1.0 5 0 EOR
%   B3:1/6  "AUXILIAR BOMBA 1 LIGADA" %
%   I:2.0/1  MT2211PSL  "PS2211 PRESSOSTATO BOMBA 1 PRESSAO BAIXA" %
%   B3:0/1  "BOMBA 1 DEFEITO" %
%   B13:1/4  ZS2212LPF  "VALV SUCCAO BOMBA 1 POSICAO FECHADO" %
%   T4:34  "TIMER LIGA PROXIMA BOMBA" %
% Rung: 7 %
% BOMBA 2 LIGADA %
SOR XIC I:2.0/4 OTE B11:2/6 EOR
%   I:2.0/4  MT2213SLIC  "MT2213 MOTOR BOMBA 2 CONTATOR FECHADO" %
%   B11:2/6  MT2213SLLI  "BOMBA 2 LIGADA" %
% Rung: 8 %
SOR BST XIC I:2.0/4 NXB XIC I:9.1/2 BND OTE O:9.5/1 EOR
%   I:2.0/4  MT2213SLIC  "MT2213 MOTOR BOMBA 2 CONTATOR FECHADO" %
%   I:9.1/2  C1BTL  "1B3MC2211 BOTAO TESTE DE LAMPADA (MESA DE COMANDO)" %
%   O:9.5/1  1H5CLIC  "LAMPADA BOMBA 2 LIGADA" %
% Rung: 9 %
% DISJUNTOR DESLIGADO %
SOR XIO I:2.0/2 OTE B13:2/1 EOR
%   I:2.0/2  "MT2213 MOTOR BOMBA 2 DISJ LIGADO" %
%   B13:2/1  MT2213SDLC  "BOMBA 2 DISJ DESLIGADO" %
% Rung: 10 %
% SOBRECARGA %
SOR XIC I:2.0/5 OTE B13:2/2 EOR
%   I:2.0/5  MT2213SSCC  "MT2213 MOTOR BOMBA 2 SOBRECARGA" %
%   B13:2/2  MT2213ASC  "BOMBA 2 SOBRECARGA" %
% Rung: 11 %
% DISJUNTOR EM TRIP %
SOR XIO I:2.0/3 OTE B13:2/3 EOR
%   I:2.0/3  "MT2213 MOTOR BOMBA 2 DISJ EM TRIP" %
%   B13:2/3  MT2213SDAT  "BOMBA 2 DISJUNTOR EM TRIP" %

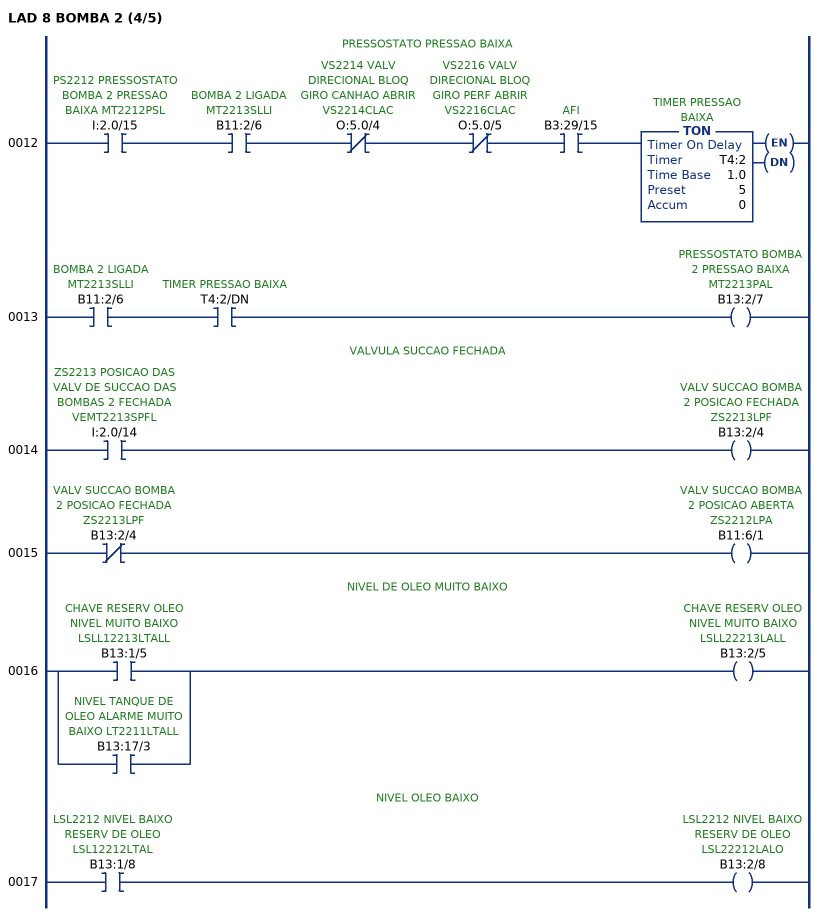
% Rung: 12 %
% PRESSOSTATO PRESSAO BAIXA %
SOR XIC I:2.0/15 XIC B11:2/6 XIO O:5.0/4 XIO O:5.0/5 XIC B3:29/15 TON T4:2 1.0 5 0 EOR
%   I:2.0/15  MT2212PSL  "PS2212 PRESSOSTATO BOMBA 2 PRESSAO BAIXA" %
%   B11:2/6  MT2213SLLI  "BOMBA 2 LIGADA" %
%   O:5.0/4  VS2214CLAC  "VS2214 VALV DIRECIONAL BLOQ GIRO CANHAO ABRIR" %
%   O:5.0/5  VS2216CLAC  "VS2216 VALV DIRECIONAL BLOQ GIRO PERF ABRIR" %
%   B3:29/15  AFI %
%   T4:2  "TIMER PRESSAO BAIXA" %
% Rung: 13 %
SOR XIC B11:2/6 XIC T4:2/DN OTE B13:2/7 EOR
%   B11:2/6  MT2213SLLI  "BOMBA 2 LIGADA" %
%   T4:2  "TIMER PRESSAO BAIXA" %
%   B13:2/7  MT2213PAL  "PRESSOSTATO BOMBA 2 PRESSAO BAIXA" %
% Rung: 14 %
% VALVULA SUCCAO FECHADA %
SOR XIC I:2.0/14 OTE B13:2/4 EOR
%   I:2.0/14  VEMT2213SPFL  "ZS2213 POSICAO DAS VALV DE SUCCAO DAS BOMBAS 2 FECHADA" %
%   B13:2/4  ZS2213LPF  "VALV SUCCAO BOMBA 2 POSICAO FECHADA" %
% Rung: 15 %
SOR XIO B13:2/4 OTE B11:6/1 EOR
%   B13:2/4  ZS2213LPF  "VALV SUCCAO BOMBA 2 POSICAO FECHADA" %
%   B11:6/1  ZS2212LPA  "VALV SUCCAO BOMBA 2 POSICAO ABERTA" %
% Rung: 16 %
% NIVEL DE OLEO MUITO BAIXO %
SOR BST XIC B13:1/5 NXB XIC B13:17/3 BND OTE B13:2/5 EOR
%   B13:1/5  LSLL12213LTALL  "CHAVE RESERV OLEO NIVEL MUITO BAIXO" %
%   B13:17/3  LT2211LTALL  "NIVEL TANQUE DE OLEO ALARME MUITO BAIXO" %
%   B13:2/5  LSLL22213LALL  "CHAVE RESERV OLEO NIVEL MUITO BAIXO" %
% Rung: 17 %
% NIVEL OLEO BAIXO %
SOR XIC B13:1/8 OTE B13:2/8 EOR
%   B13:1/8  LSL12212LTAL  "LSL2212 NIVEL BAIXO RESERV DE OLEO" %
%   B13:2/8  LSL22212LALO  "LSL2212 NIVEL BAIXO RESERV DE OLEO" %

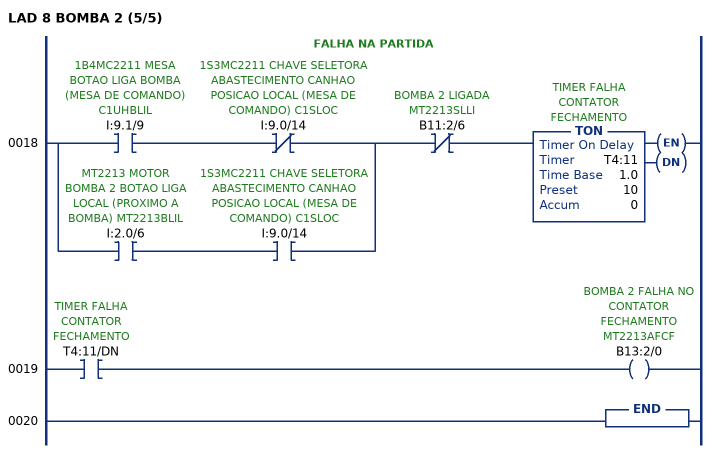
% Rung: 18 %
% TITLE: FALHA NA PARTIDA %
SOR BST XIC I:9.1/9 XIO I:9.0/14 NXB XIC I:2.0/6 XIC I:9.0/14 BND XIO B11:2/6 TON T4:11 1.0 10 0 EOR
%   I:9.1/9  C1UHBLIL  "1B4MC2211 MESA BOTAO LIGA BOMBA (MESA DE COMANDO)" %
%   I:9.0/14  C1SLOC  "1S3MC2211 CHAVE SELETORA ABASTECIMENTO CANHAO POSICAO LOCAL (MESA DE COMANDO)" %
%   I:2.0/6  MT2213BLIL  "MT2213 MOTOR BOMBA 2 BOTAO LIGA LOCAL (PROXIMO A BOMBA)" %
%   B11:2/6  MT2213SLLI  "BOMBA 2 LIGADA" %
%   T4:11  "TIMER FALHA CONTATOR FECHAMENTO" %
% Rung: 19 %
SOR XIC T4:11/DN OTE B13:2/0 EOR
%   T4:11/DN  "TIMER FALHA CONTATOR FECHAMENTO" %
%   B13:2/0  MT2213AFCF  "BOMBA 2 FALHA NO CONTATOR FECHAMENTO" %
% Rung: 20 %
SOR END EOR

LADDER 9 "BOMBA REF"    % Bomba Refrigeracao 1 %
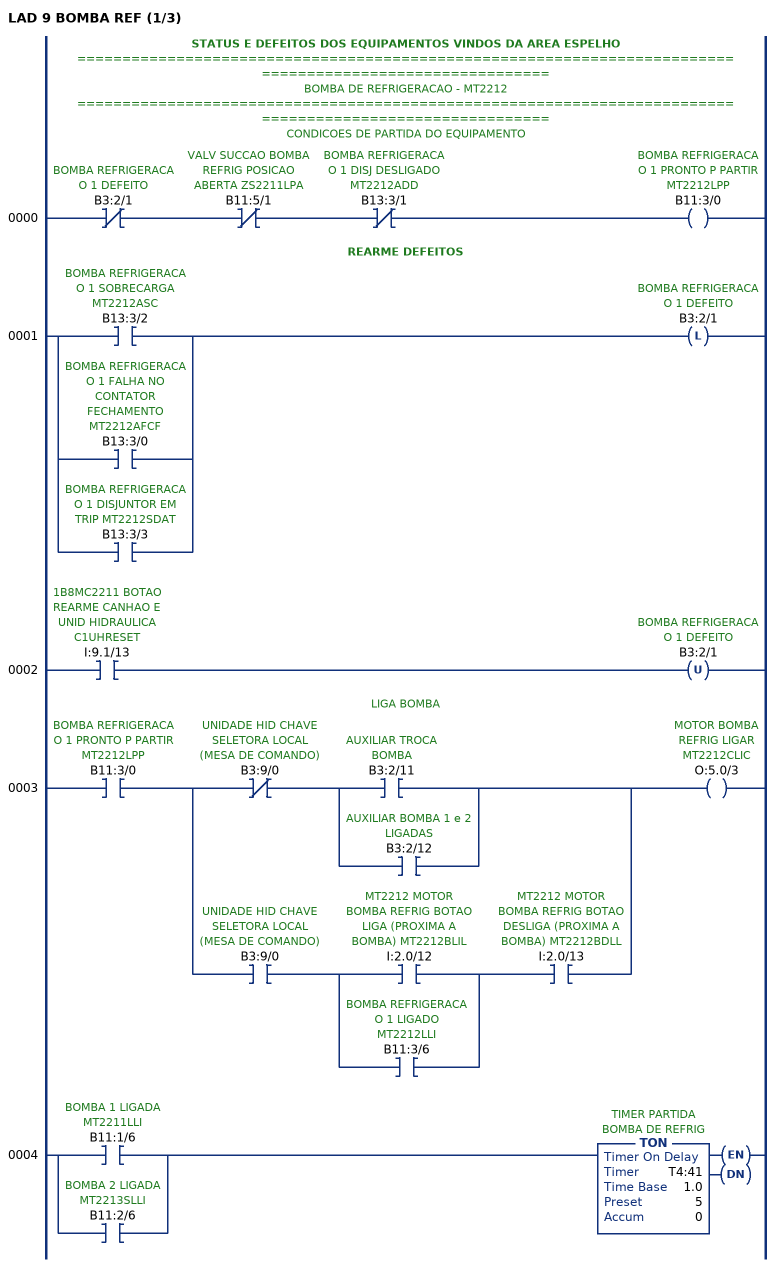
% Rung: 0 %
% TITLE: STATUS E DEFEITOS DOS EQUIPAMENTOS VINDOS DA AREA ESPELHO %
% =========================================================================================================
% BOMBA DE REFRIGERACAO - MT2212
% =========================================================================================================
% 
% CONDICOES DE PARTIDA DO EQUIPAMENTO %
SOR XIO B3:2/1 XIO B11:5/1 XIO B13:3/1 OTE B11:3/0 EOR
%   B3:2/1  "BOMBA REFRIGERACAO 1 DEFEITO" %
%   B11:5/1  ZS2211LPA  "VALV SUCCAO BOMBA REFRIG POSICAO ABERTA" %
%   B13:3/1  MT2212ADD  "BOMBA REFRIGERACAO 1 DISJ DESLIGADO" %
%   B11:3/0  MT2212LPP  "BOMBA REFRIGERACAO 1 PRONTO P PARTIR" %
% Rung: 1 %
% TITLE: REARME DEFEITOS %
SOR BST XIC B13:3/2 NXB XIC B13:3/0 NXB XIC B13:3/3 BND OTL B3:2/1 EOR
%   B13:3/2  MT2212ASC  "BOMBA REFRIGERACAO 1 SOBRECARGA" %
%   B13:3/0  MT2212AFCF  "BOMBA REFRIGERACAO 1 FALHA NO CONTATOR FECHAMENTO" %
%   B13:3/3  MT2212SDAT  "BOMBA REFRIGERACAO 1 DISJUNTOR EM TRIP" %
%   B3:2/1  "BOMBA REFRIGERACAO 1 DEFEITO" %
% Rung: 2 %
SOR XIC I:9.1/13 OTU B3:2/1 EOR
%   I:9.1/13  C1UHRESET  "1B8MC2211 BOTAO REARME CANHAO E UNID HIDRAULICA" %
%   B3:2/1  "BOMBA REFRIGERACAO 1 DEFEITO" %
% Rung: 3 %
% LIGA BOMBA %
SOR XIC B11:3/0 BST XIO B3:9/0 BST XIC B3:2/11 NXB XIC B3:2/12 BND NXB XIC B3:9/0 BST XIC I:2.0/12 NXB XIC B11:3/6 BND XIC I:2.0/13 BND OTE O:5.0/3 EOR
%   B11:3/0  MT2212LPP  "BOMBA REFRIGERACAO 1 PRONTO P PARTIR" %
%   B3:9/0  "UNIDADE HID CHAVE SELETORA LOCAL (MESA DE COMANDO)" %
%   B3:2/11  "AUXILIAR TROCA BOMBA" %
%   B3:2/12  "AUXILIAR BOMBA 1 e 2 LIGADAS" %
%   I:2.0/12  MT2212BLIL  "MT2212 MOTOR BOMBA REFRIG BOTAO LIGA (PROXIMA A BOMBA)" %
%   B11:3/6  MT2212LLI  "BOMBA REFRIGERACAO 1 LIGADO" %
%   I:2.0/13  MT2212BDLL  "MT2212 MOTOR BOMBA REFRIG BOTAO DESLIGA (PROXIMA A BOMBA)" %
%   O:5.0/3  MT2212CLIC  "MOTOR BOMBA REFRIG LIGAR" %
% Rung: 4 %
SOR BST XIC B11:1/6 NXB XIC B11:2/6 BND TON T4:41 1.0 5 0 EOR
%   B11:1/6  MT2211LLI  "BOMBA 1 LIGADA" %
%   B11:2/6  MT2213SLLI  "BOMBA 2 LIGADA" %
%   T4:41  "TIMER PARTIDA BOMBA DE REFRIG" %

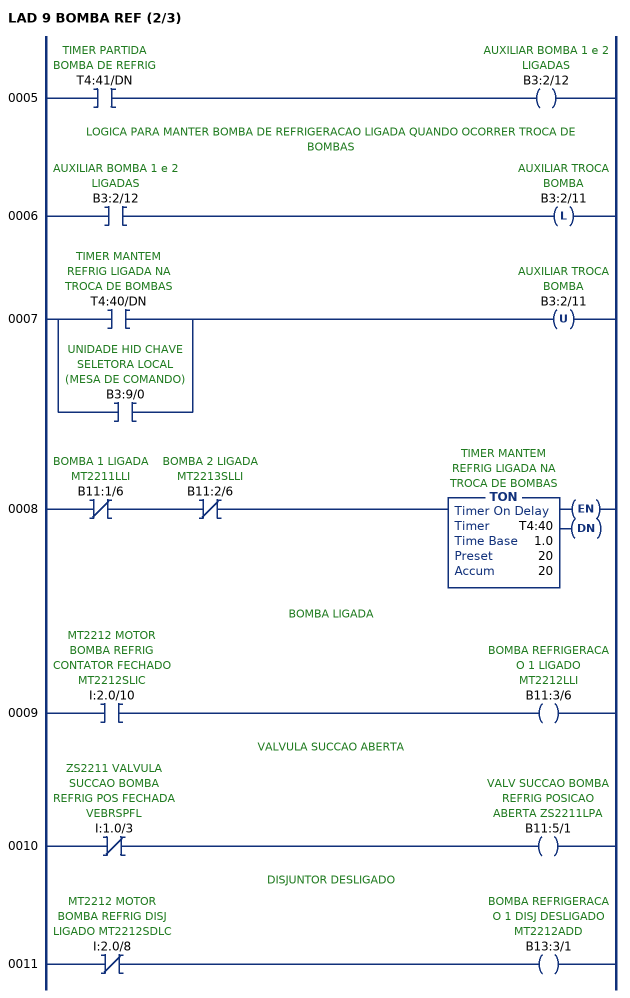
% Rung: 5 %
SOR XIC T4:41/DN OTE B3:2/12 EOR
%   T4:41  "TIMER PARTIDA BOMBA DE REFRIG" %
%   B3:2/12  "AUXILIAR BOMBA 1 e 2 LIGADAS" %
% Rung: 6 %
% LOGICA PARA MANTER BOMBA DE REFRIGERACAO LIGADA QUANDO OCORRER TROCA DE BOMBAS %
SOR XIC B3:2/12 OTL B3:2/11 EOR
%   B3:2/12  "AUXILIAR BOMBA 1 e 2 LIGADAS" %
%   B3:2/11  "AUXILIAR TROCA BOMBA" %
% Rung: 7 %
SOR BST XIC T4:40/DN NXB XIC B3:9/0 BND OTU B3:2/11 EOR
%   T4:40  "TIMER MANTEM REFRIG LIGADA NA TROCA DE BOMBAS" %
%   B3:9/0  "UNIDADE HID CHAVE SELETORA LOCAL (MESA DE COMANDO)" %
%   B3:2/11  "AUXILIAR TROCA BOMBA" %
% Rung: 8 %
SOR XIO B11:1/6 XIO B11:2/6 TON T4:40 1.0 20 20 EOR
%   B11:1/6  MT2211LLI  "BOMBA 1 LIGADA" %
%   B11:2/6  MT2213SLLI  "BOMBA 2 LIGADA" %
%   T4:40  "TIMER MANTEM REFRIG LIGADA NA TROCA DE BOMBAS" %
% Rung: 9 %
% BOMBA LIGADA %
SOR XIC I:2.0/10 OTE B11:3/6 EOR
%   I:2.0/10  MT2212SLIC  "MT2212 MOTOR BOMBA REFRIG CONTATOR FECHADO" %
%   B11:3/6  MT2212LLI  "BOMBA REFRIGERACAO 1 LIGADO" %
% Rung: 10 %
% VALVULA SUCCAO ABERTA %
SOR XIO I:1.0/3 OTE B11:5/1 EOR
%   I:1.0/3  VEBRSPFL  "ZS2211 VALVULA SUCCAO BOMBA REFRIG POS FECHADA" %
%   B11:5/1  ZS2211LPA  "VALV SUCCAO BOMBA REFRIG POSICAO ABERTA" %
% Rung: 11 %
% DISJUNTOR DESLIGADO %
SOR XIO I:2.0/8 OTE B13:3/1 EOR
%   I:2.0/8  MT2212SDLC  "MT2212 MOTOR BOMBA REFRIG DISJ LIGADO" %
%   B13:3/1  MT2212ADD  "BOMBA REFRIGERACAO 1 DISJ DESLIGADO" %

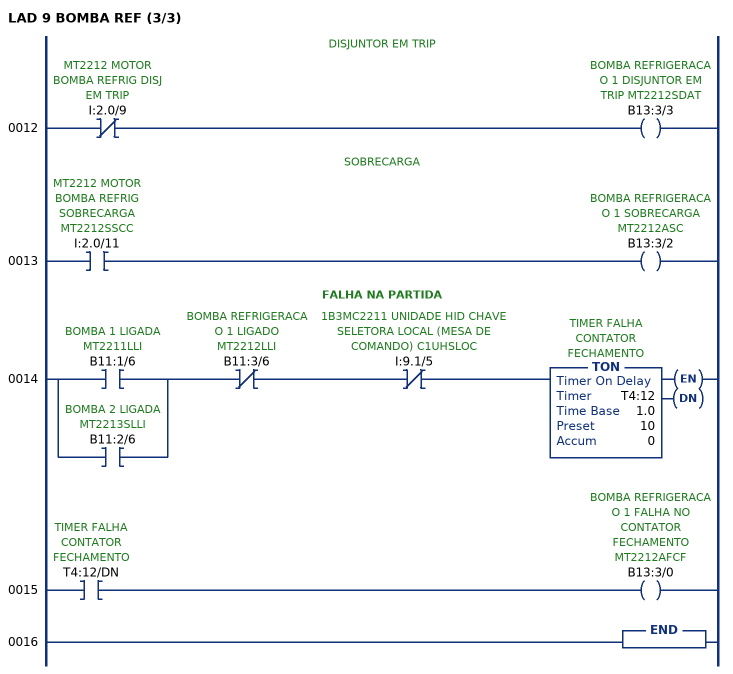
% Rung: 12 %
% DISJUNTOR EM TRIP %
SOR XIO I:2.0/9 OTE B13:3/3 EOR
%   I:2.0/9  "MT2212 MOTOR BOMBA REFRIG DISJ EM TRIP" %
%   B13:3/3  MT2212SDAT  "BOMBA REFRIGERACAO 1 DISJUNTOR EM TRIP" %
% Rung: 13 %
% SOBRECARGA %
SOR XIC I:2.0/11 OTE B13:3/2 EOR
%   I:2.0/11  MT2212SSCC  "MT2212 MOTOR BOMBA REFRIG SOBRECARGA" %
%   B13:3/2  MT2212ASC  "BOMBA REFRIGERACAO 1 SOBRECARGA" %
% Rung: 14 %
% TITLE: FALHA NA PARTIDA %
SOR BST XIC B11:1/6 NXB XIC B11:2/6 BND XIO B11:3/6 XIO I:9.1/5 TON T4:12 1.0 10 0 EOR
%   B11:1/6  MT2211LLI  "BOMBA 1 LIGADA" %
%   B11:2/6  MT2213SLLI  "BOMBA 2 LIGADA" %
%   B11:3/6  MT2212LLI  "BOMBA REFRIGERACAO 1 LIGADO" %
%   I:9.1/5  C1UHSLOC  "1B3MC2211 UNIDADE HID CHAVE SELETORA LOCAL (MESA DE COMANDO)" %
%   T4:12  "TIMER FALHA CONTATOR FECHAMENTO" %
% Rung: 15 %
SOR XIC T4:12/DN OTE B13:3/0 EOR
%   T4:12  "TIMER FALHA CONTATOR FECHAMENTO" %
%   B13:3/0  MT2212AFCF  "BOMBA REFRIGERACAO 1 FALHA NO CONTATOR FECHAMENTO" %
% Rung: 16 %
SOR END EOR

LADDER 11 "PRESS INJ"    % Pressao de injecao mais alta %
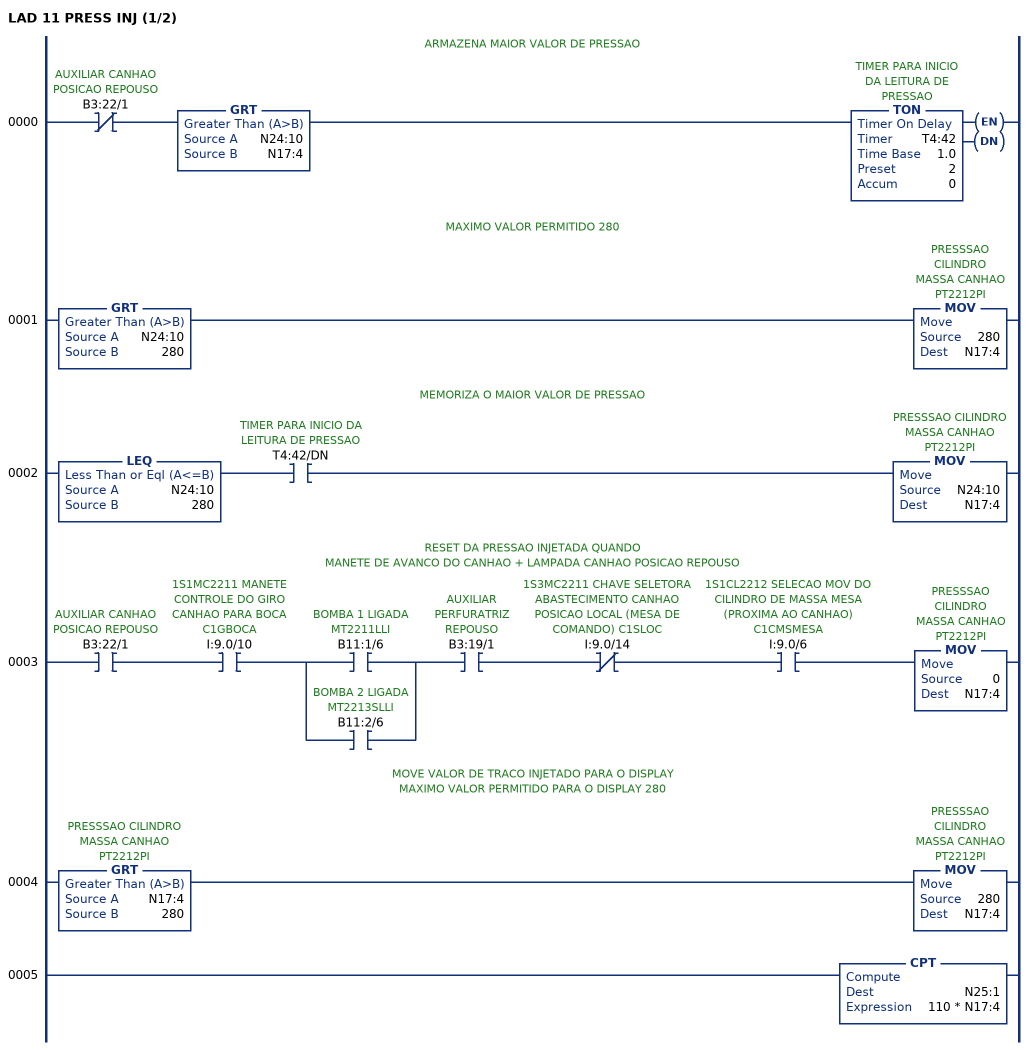
% Rung: 0 %
% ARMAZENA MAIOR VALOR DE PRESSAO %
SOR XIO B3:22/1 GRT N24:10 N17:4 TON T4:42 1.0 2 0 EOR
%   B3:22/1  "AUXILIAR CANHAO POSICAO REPOUSO" %
%   N17:4  PT2212PI  "PRESSSAO CILINDRO MASSA CANHAO" %
%   T4:42  "TIMER PARA INICIO DA LEITURA DE PRESSAO" %
% Rung: 1 %
% MAXIMO VALOR PERMITIDO 280 %
SOR GRT N24:10 280 MOV 280 N17:4 EOR
%   N17:4  PT2212PI  "PRESSSAO CILINDRO MASSA CANHAO" %
% Rung: 2 %
% MEMORIZA O MAIOR VALOR DE PRESSAO %
SOR LEQ N24:10 280 XIC T4:42/DN MOV N24:10 N17:4 EOR
%   T4:42  "TIMER PARA INICIO DA LEITURA DE PRESSAO" %
%   N17:4  PT2212PI  "PRESSSAO CILINDRO MASSA CANHAO" %
% Rung: 3 %
% RESET DA PRESSAO INJETADA QUANDO
% MANETE DE AVANCO DO CANHAO + LAMPADA CANHAO POSICAO REPOUSO %
SOR XIC B3:22/1 XIC I:9.0/10 BST XIC B11:1/6 NXB XIC B11:2/6 BND XIC B3:19/1 XIO I:9.0/14 XIC I:9.0/6 MOV 0 N17:4 EOR
%   B3:22/1  "AUXILIAR CANHAO POSICAO REPOUSO" %
%   I:9.0/10  C1GBOCA  "1S1MC2211 MANETE CONTROLE DO GIRO CANHAO PARA BOCA" %
%   B11:1/6  MT2211LLI  "BOMBA 1 LIGADA" %
%   B11:2/6  MT2213SLLI  "BOMBA 2 LIGADA" %
%   B3:19/1  "AUXILIAR PERFURATRIZ REPOUSO" %
%   I:9.0/14  C1SLOC  "1S3MC2211 CHAVE SELETORA ABASTECIMENTO CANHAO POSICAO LOCAL (MESA DE COMANDO)" %
%   I:9.0/6  C1CMSMESA  "1S1CL2212 SELECAO MOV DO CILINDRO DE MASSA MESA (PROXIMA AO CANHAO)" %
%   N17:4  PT2212PI  "PRESSSAO CILINDRO MASSA CANHAO" %
% Rung: 4 %
% MOVE VALOR DE TRACO INJETADO PARA O DISPLAY
% MAXIMO VALOR PERMITIDO PARA O DISPLAY 280 %
SOR GRT N17:4 280 MOV 280 N17:4 EOR
%   N17:4  PT2212PI  "PRESSSAO CILINDRO MASSA CANHAO" %
% Rung: 5 %
SOR CPT N25:1 " 110 * N17:4 " EOR
%   N17:4  PT2212PI  "PRESSSAO CILINDRO MASSA CANHAO" %

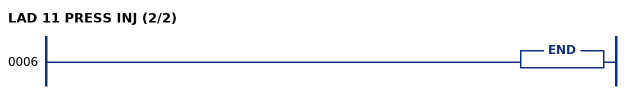
% Rung: 6 %
SOR END EOR

LADDER 12 "TRACO INJ"    % Volume Lama Injetado %
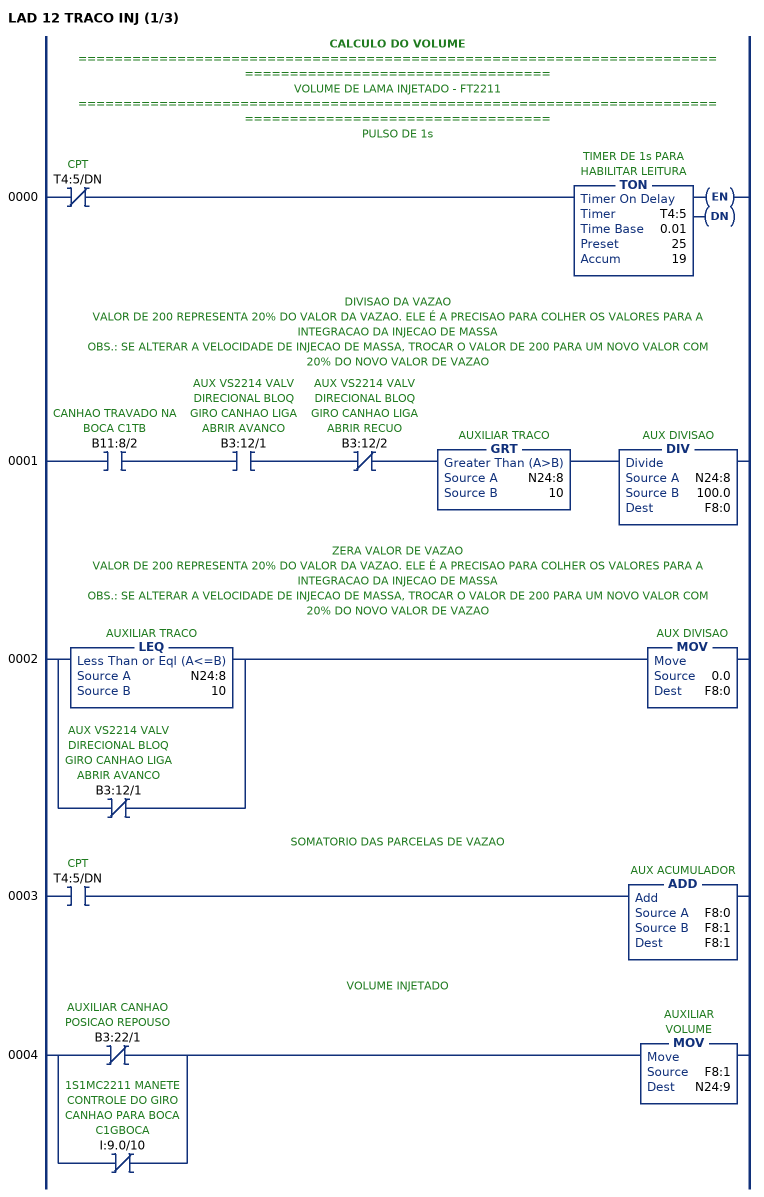
% Rung: 0 %
% TITLE: CALCULO DO VOLUME %
% =========================================================================================================
% VOLUME DE LAMA INJETADO - FT2211
% =========================================================================================================
% PULSO DE 1s %
SOR XIO T4:5/DN TON T4:5 0.01 25 19 EOR
%   T4:5/DN  CPT %
%   T4:5  "TIMER DE 1s PARA HABILITAR LEITURA" %
% Rung: 1 %
% DIVISAO DA VAZAO
% VALOR DE 200 REPRESENTA 20% DO VALOR DA VAZAO. ELE É A PRECISAO PARA COLHER OS VALORES PARA A INTEGRACAO DA INJECAO DE MASSA
% OBS.: SE ALTERAR A VELOCIDADE DE INJECAO DE MASSA, TROCAR O VALOR DE 200 PARA UM NOVO VALOR COM 20% DO NOVO VALOR DE VAZAO %
SOR XIC B11:8/2 XIC B3:12/1 XIO B3:12/2 GRT N24:8 10 DIV N24:8 100.0 F8:0 EOR
%   B11:8/2  C1TB  "CANHAO TRAVADO NA BOCA" %
%   B3:12/1  "AUX VS2214 VALV DIRECIONAL BLOQ GIRO CANHAO LIGA ABRIR AVANCO" %
%   B3:12/2  "AUX VS2214 VALV DIRECIONAL BLOQ GIRO CANHAO LIGA ABRIR RECUO" %
%   N24:8  "AUXILIAR TRACO" %
%   F8:0  "AUX DIVISAO" %
% Rung: 2 %
% ZERA VALOR DE VAZAO
% VALOR DE 200 REPRESENTA 20% DO VALOR DA VAZAO. ELE É A PRECISAO PARA COLHER OS VALORES PARA A INTEGRACAO DA INJECAO DE MASSA
% OBS.: SE ALTERAR A VELOCIDADE DE INJECAO DE MASSA, TROCAR O VALOR DE 200 PARA UM NOVO VALOR COM 20% DO NOVO VALOR DE VAZAO %
SOR BST LEQ N24:8 10 NXB XIO B3:12/1 BND MOV 0.0 F8:0 EOR
%   N24:8  "AUXILIAR TRACO" %
%   B3:12/1  "AUX VS2214 VALV DIRECIONAL BLOQ GIRO CANHAO LIGA ABRIR AVANCO" %
%   F8:0  "AUX DIVISAO" %
% Rung: 3 %
% SOMATORIO DAS PARCELAS DE VAZAO %
SOR XIC T4:5/DN ADD F8:0 F8:1 F8:1 EOR
%   T4:5/DN  CPT %
%   F8:0  "AUX DIVISAO" %
%   F8:1  "AUX ACUMULADOR" %
% Rung: 4 %
% VOLUME INJETADO %
SOR BST XIO B3:22/1 NXB XIO I:9.0/10 BND MOV F8:1 N24:9 EOR
%   B3:22/1  "AUXILIAR CANHAO POSICAO REPOUSO" %
%   I:9.0/10  C1GBOCA  "1S1MC2211 MANETE CONTROLE DO GIRO CANHAO PARA BOCA" %
%   F8:1  "AUX ACUMULADOR" %
%   N24:9  "AUXILIAR VOLUME" %

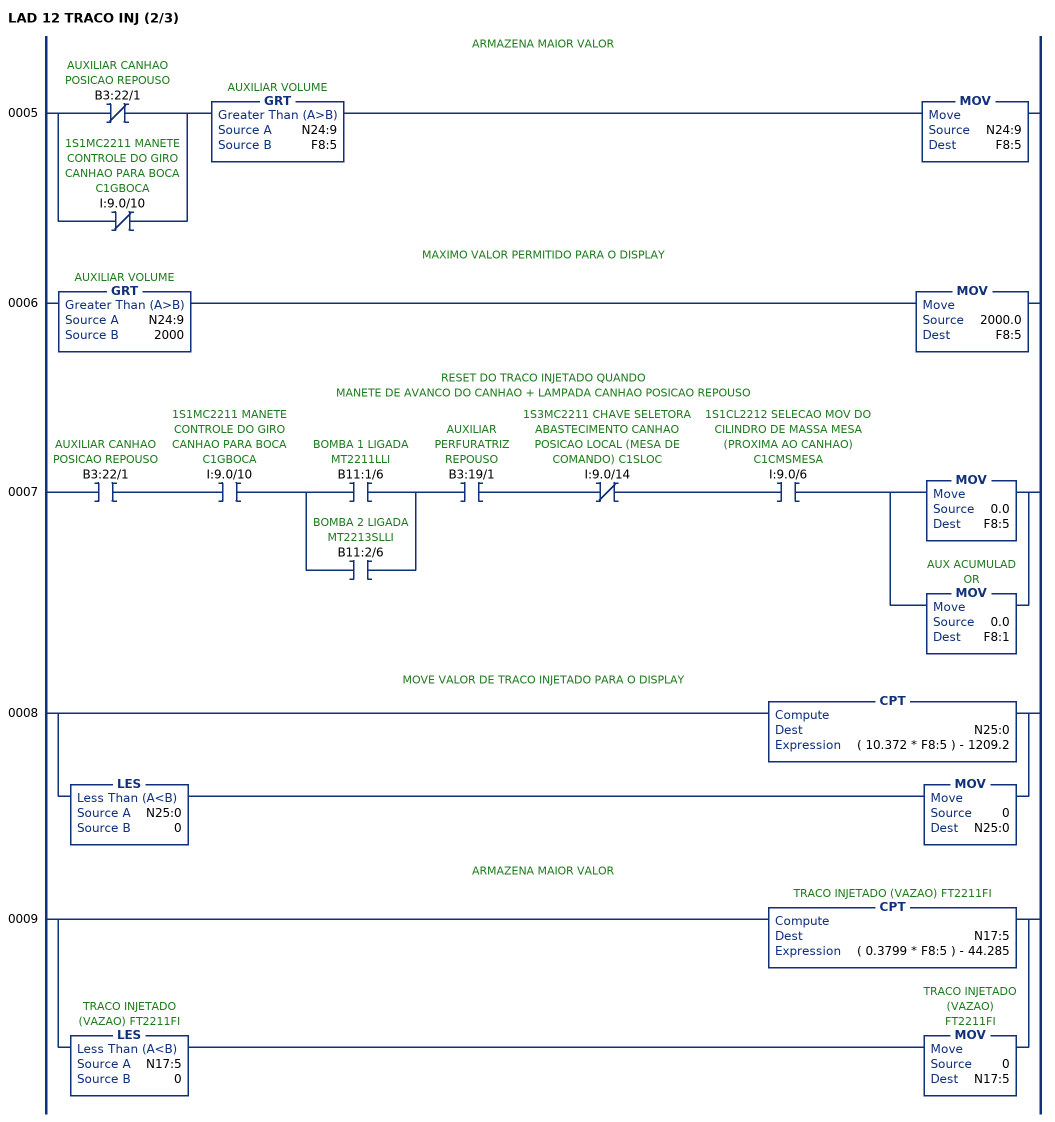
% Rung: 5 %
% ARMAZENA MAIOR VALOR %
SOR BST XIO B3:22/1 NXB XIO I:9.0/10 BND GRT N24:9 F8:5 MOV N24:9 F8:5 EOR
%   B3:22/1  "AUXILIAR CANHAO POSICAO REPOUSO" %
%   I:9.0/10  C1GBOCA  "1S1MC2211 MANETE CONTROLE DO GIRO CANHAO PARA BOCA" %
%   N24:9  "AUXILIAR VOLUME" %
% Rung: 6 %
% MAXIMO VALOR PERMITIDO PARA O DISPLAY %
SOR GRT N24:9 2000 MOV 2000.0 F8:5 EOR
%   N24:9  "AUXILIAR VOLUME" %
% Rung: 7 %
% RESET DO TRACO INJETADO QUANDO
% MANETE DE AVANCO DO CANHAO + LAMPADA CANHAO POSICAO REPOUSO %
SOR XIC B3:22/1 XIC I:9.0/10 BST XIC B11:1/6 NXB XIC B11:2/6 BND XIC B3:19/1 XIO I:9.0/14 XIC I:9.0/6 BST MOV 0.0 F8:5 NXB MOV 0.0 F8:1 BND EOR
%   B3:22/1  "AUXILIAR CANHAO POSICAO REPOUSO" %
%   I:9.0/10  C1GBOCA  "1S1MC2211 MANETE CONTROLE DO GIRO CANHAO PARA BOCA" %
%   B11:1/6  MT2211LLI  "BOMBA 1 LIGADA" %
%   B11:2/6  MT2213SLLI  "BOMBA 2 LIGADA" %
%   B3:19/1  "AUXILIAR PERFURATRIZ REPOUSO" %
%   I:9.0/14  C1SLOC  "1S3MC2211 CHAVE SELETORA ABASTECIMENTO CANHAO POSICAO LOCAL (MESA DE COMANDO)" %
%   I:9.0/6  C1CMSMESA  "1S1CL2212 SELECAO MOV DO CILINDRO DE MASSA MESA (PROXIMA AO CANHAO)" %
%   F8:1  "AUX ACUMULADOR" %
% Rung: 8 %
% MOVE VALOR DE TRACO INJETADO PARA O DISPLAY %
SOR BST CPT N25:0 " ( 10.372 * F8:5 ) - 1209.2 " NXB LES N25:0 0 MOV 0 N25:0 BND EOR
% Rung: 9 %
% ARMAZENA MAIOR VALOR %
SOR BST CPT N17:5 " ( 0.3799 * F8:5 ) - 44.285 " NXB LES N17:5 0 MOV 0 N17:5 BND EOR
%   N17:5  FT2211FI  "TRACO INJETADO (VAZAO)" %

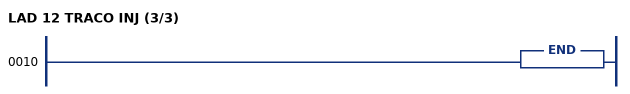
% Rung: 10 %
SOR END EOR

LADDER 13 "CANHAO"    % Controle do Giro do Canhao %
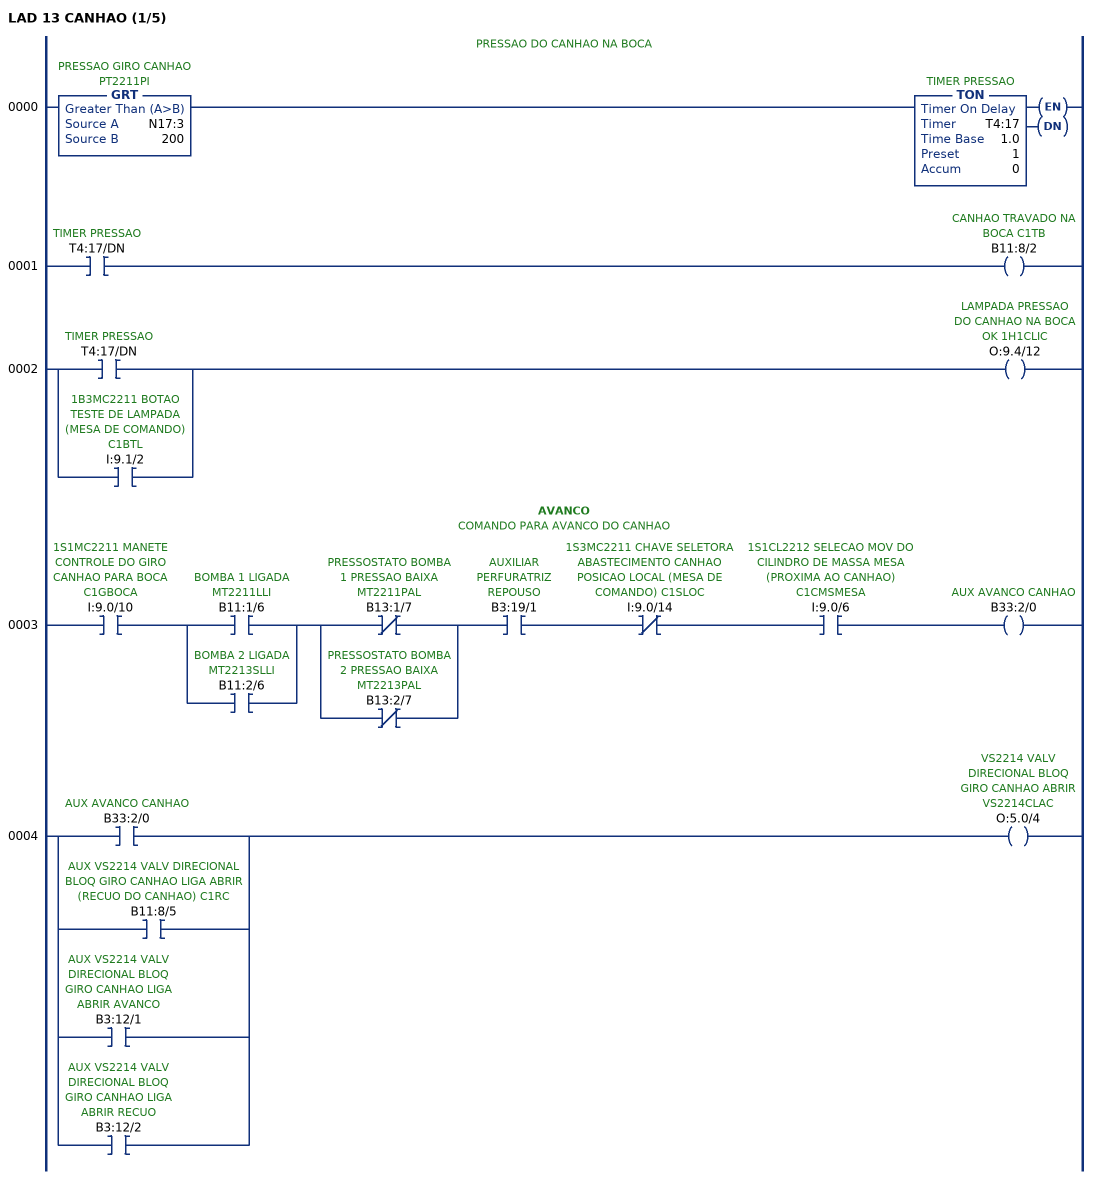
% Rung: 0 %
% PRESSAO DO CANHAO NA BOCA %
SOR GRT N17:3 200 TON T4:17 1.0 1 0 EOR
%   N17:3  PT2211PI  "PRESSAO GIRO CANHAO" %
%   T4:17  "TIMER PRESSAO" %
% Rung: 1 %
SOR XIC T4:17/DN OTE B11:8/2 EOR
%   T4:17  "TIMER PRESSAO" %
%   B11:8/2  C1TB  "CANHAO TRAVADO NA BOCA" %
% Rung: 2 %
SOR BST XIC T4:17/DN NXB XIC I:9.1/2 BND OTE O:9.4/12 EOR
%   T4:17  "TIMER PRESSAO" %
%   I:9.1/2  C1BTL  "1B3MC2211 BOTAO TESTE DE LAMPADA (MESA DE COMANDO)" %
%   O:9.4/12  1H1CLIC  "LAMPADA PRESSAO DO CANHAO NA BOCA OK" %
% Rung: 3 %
% TITLE: AVANCO %
% COMANDO PARA AVANCO DO CANHAO %
SOR XIC I:9.0/10 BST XIC B11:1/6 NXB XIC B11:2/6 BND BST XIO B13:1/7 NXB XIO B13:2/7 BND XIC B3:19/1 XIO I:9.0/14 XIC I:9.0/6 OTE B33:2/0 EOR
%   I:9.0/10  C1GBOCA  "1S1MC2211 MANETE CONTROLE DO GIRO CANHAO PARA BOCA" %
%   B11:1/6  MT2211LLI  "BOMBA 1 LIGADA" %
%   B11:2/6  MT2213SLLI  "BOMBA 2 LIGADA" %
%   B13:1/7  MT2211PAL  "PRESSOSTATO BOMBA 1 PRESSAO BAIXA" %
%   B13:2/7  MT2213PAL  "PRESSOSTATO BOMBA 2 PRESSAO BAIXA" %
%   B3:19/1  "AUXILIAR PERFURATRIZ REPOUSO" %
%   I:9.0/14  C1SLOC  "1S3MC2211 CHAVE SELETORA ABASTECIMENTO CANHAO POSICAO LOCAL (MESA DE COMANDO)" %
%   I:9.0/6  C1CMSMESA  "1S1CL2212 SELECAO MOV DO CILINDRO DE MASSA MESA (PROXIMA AO CANHAO)" %
%   B33:2/0  "AUX AVANCO CANHAO" %
% Rung: 4 %
SOR BST XIC B33:2/0 NXB XIC B11:8/5 NXB XIC B3:12/1 NXB XIC B3:12/2 BND OTE O:5.0/4 EOR
%   B33:2/0  "AUX AVANCO CANHAO" %
%   B11:8/5  C1RC  "AUX VS2214 VALV DIRECIONAL BLOQ GIRO CANHAO LIGA ABRIR (RECUO DO CANHAO)" %
%   B3:12/1  "AUX VS2214 VALV DIRECIONAL BLOQ GIRO CANHAO LIGA ABRIR AVANCO" %
%   B3:12/2  "AUX VS2214 VALV DIRECIONAL BLOQ GIRO CANHAO LIGA ABRIR RECUO" %
%   O:5.0/4  VS2214CLAC  "VS2214 VALV DIRECIONAL BLOQ GIRO CANHAO ABRIR" %

